KUKA KRL program: MyProgram_123().src

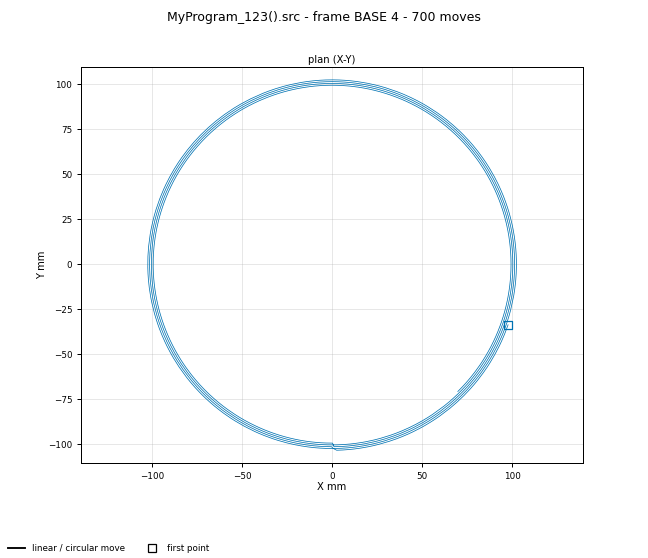
[picture p0: tool path of MyProgram_123().src in frame BASE 4, 700 of 700 moves have a stored position in this frame; points joined in program order, loops and branches not executed]
&ACCESS RVP
&REL 1
&PARAM TEMPLATE = C:\KRC\Roboter\Template\vorgabe
&PARAM EDITMASK = *
DEF MyProgram_123()
; ---- Setting reference (Base) ----
$BASE = BASE_DATA[4]

; --------------------------
; ---- Setting tool (TCP) ----
$TOOL = TOOL_DATA[3]
; --------------------------

$VEL.CP = VEL_APROX_PRINT
Startdeposition()
$VEL.CP = VEL_PRINT
LIN {X 97.6881,Y -33.6698,Z 103,A -23.787,B 24.9383,C -1.8145,E1 25.1507,E2 469.3571} C_DIS
LIN {X 95.781,Y -38.76,Z 103,A -26.6465,B 24.9385,C -1.8116,E1 25.1479,E2 472.2074} C_DIS
LIN {X 94.2157,Y -42.4228,Z 103,A -28.8922,B 24.939,C -1.8033,E1 25.1453,E2 474.4605} C_DIS
LIN {X 93.0003,Y -45.0257,Z 103,A -30.4605,B 24.9393,C -1.7995,E1 25.1435,E2 476.0292} C_DIS
LIN {X 90.4664,Y -49.9238,Z 103,A -33.4281,B 24.9397,C -1.7942,E1 25.1396,E2 478.9937} C_DIS
LIN {X 87.7675,Y -54.5272,Z 103,A -36.2353,B 24.9398,C -1.7919,E1 25.1357,E2 481.7919} C_DIS
LIN {X 86.0982,Y -57.1268,Z 103,A -37.9177,B 24.9401,C -1.7883,E1 25.1331,E2 483.4744} C_DIS
LIN {X 83.9825,Y -60.1936,Z 103,A -41.1362,B 24.9436,C -1.7353,E1 25.1277,E2 486.8023} C_DIS
LIN {X 80.9511,Y -64.2124,Z 103,A -42.7215,B 24.9408,C -1.7771,E1 25.1252,E2 488.2813} C_DIS
LIN {X 79.0718,Y -66.5134,Z 103,A -44.9977,B 24.9428,C -1.7469,E1 25.121,E2 490.6184} C_DIS
LIN {X 76.8006,Y -69.1233,Z 103,A -47.4937,B 24.9447,C -1.7186,E1 25.1163,E2 493.1703} C_DIS
LIN {X 73.2293,Y -72.8966,Z 103,A -49.516,B 24.9428,C -1.7463,E1 25.1125,E2 495.1185} C_DIS
LIN {X 69.1425,Y -76.7834,Z 103,A -52.3279,B 24.9425,C -1.7518,E1 25.1068,E2 497.9058} C_DIS
LIN {X 65.4366,Y -79.9649,Z 103,A -55.2445,B 24.9434,C -1.7371,E1 25.1005,E2 500.8457} C_DIS
LIN {X 59.791,Y -84.2698,Z 103,A -59.6873,B 24.9453,C -1.7083,E1 25.0905,E2 505.3406} C_DIS
LIN {X 56.834,Y -86.2913,Z 103,A -61.1986,B 24.9443,C -1.7235,E1 25.087,E2 506.811} C_DIS
LIN {X 54.8773,Y -87.5488,Z 103,A -63.0884,B 24.946,C -1.697,E1 25.0824,E2 508.7576} C_DIS
LIN {X 51.3153,Y -89.6831,Z 103,A -64.9043,B 24.9451,C -1.7122,E1 25.0781,E2 510.5318} C_DIS
LIN {X 48.7655,Y -91.0963,Z 103,A -67.0748,B 24.9466,C -1.6873,E1 25.0727,E2 512.7551} C_DIS
LIN {X 44.8398,Y -93.0897,Z 103,A -68.7427,B 24.9449,C -1.7142,E1 25.0687,E2 514.3551} C_DIS
LIN {X 42.065,Y -94.3769,Z 103,A -70.4455,B 24.9451,C -1.7113,E1 25.0643,E2 516.0605} C_DIS
LIN {X 38.6683,Y -95.8183,Z 103,A -72.4301,B 24.9451,C -1.7107,E1 25.0592,E2 518.0417} C_DIS
LIN {X 35.7045,Y -96.9617,Z 103,A -74.1219,B 24.9451,C -1.7111,E1 25.0548,E2 519.7289} C_DIS
LIN {X 31.6622,Y -98.3555,Z 103,A -76.9185,B 24.9464,C -1.6913,E1 25.0473,E2 522.567} C_DIS
LIN {X 25.8035,Y -100.0524,Z 103,A -79.9686,B 24.9458,C -1.7007,E1 25.0392,E2 525.5899} C_DIS
LIN {X 23.0245,Y -100.7284,Z 103,A -81.6681,B 24.9462,C -1.6947,E1 25.0345,E2 527.3012} C_DIS
LIN {X 20.0098,Y -101.3712,Z 103,A -83.5475,B 24.9467,C -1.6865,E1 25.0293,E2 529.1976} C_DIS
LIN {X 15.782,Y -102.1137,Z 103,A -85.6605,B 24.9461,C -1.6952,E1 25.0236,E2 531.288} C_DIS
LIN {X 12.1927,Y -102.6044,Z 103,A -87.6248,B 24.9461,C -1.6956,E1 25.0181,E2 533.2496} C_DIS
LIN {X 9.3968,Y -102.898,Z 103,A -89.2294,B 24.9463,C -1.693,E1 25.0136,E2 534.8595} C_DIS
LIN {X 5.8711,Y -103.1593,Z 103,A -91.1468,B 24.9463,C -1.6938,E1 25.0083,E2 536.7742} C_DIS
LIN {X 2.5701,Y -103.2946,Z 103,A -93.23,B 24.9469,C -1.6835,E1 25.0024,E2 538.8813} C_DIS
LIN {X 2.5701,Y -103.2946,Z 103,A -93.23,B 24.9469,C -1.6835,E1 25.0024,E2 538.8813} C_DIS
Enddeposition()
LIN {X 0.6764,Y -102.3239,Z 103,A -92.9796,B 24.9425,C -1.7511,E1 25.0036,E2 538.4707} C_DIS
Startdeposition()
$VEL.CP = VEL_PRINT
LIN {X 5.1299,Y -102.2014,Z 103,A -90.7138,B 24.9431,C -1.743,E1 25.0098,E2 536.2248} C_DIS
LIN {X 8.6252,Y -101.9657,Z 103,A -88.8428,B 24.9432,C -1.7404,E1 25.015,E2 534.3608} C_DIS
LIN {X 11.7328,Y -101.654,Z 103,A -87.1009,B 24.9432,C -1.7411,E1 25.0199,E2 532.6184} C_DIS
LIN {X 14.8311,Y -101.2492,Z 103,A -85.4205,B 24.9432,C -1.7396,E1 25.0245,E2 530.9431} C_DIS
LIN {X 18.0457,Y -100.725,Z 103,A -82.9702,B 24.9416,C -1.7658,E1 25.0314,E2 528.4332} C_DIS
LIN {X 21.7381,Y -99.9932,Z 103,A -81.7936,B 24.9439,C -1.7308,E1 25.0344,E2 527.341} C_DIS
LIN {X 25.3407,Y -99.1415,Z 103,A -78.7726,B 24.9412,C -1.7705,E1 25.0428,E2 524.2304} C_DIS
LIN {X 29.0621,Y -98.1151,Z 103,A -77.3225,B 24.943,C -1.7445,E1 25.0466,E2 522.8443} C_DIS
LIN {X 34.35,Y -96.3924,Z 103,A -74.2269,B 24.9428,C -1.7476,E1 25.0548,E2 519.7474} C_DIS
LIN {X 36.8204,Y -95.4766,Z 103,A -72.3941,B 24.9417,C -1.7639,E1 25.0596,E2 517.8799} C_DIS
LIN {X 40.9607,Y -93.7731,Z 103,A -70.1365,B 24.9421,C -1.7576,E1 25.0654,E2 515.6426} C_DIS
LIN {X 44.2148,Y -92.2835,Z 103,A -67.2701,B 24.9396,C -1.7958,E1 25.0728,E2 512.6934} C_DIS
LIN {X 48.6188,Y -90.0412,Z 103,A -65.4434,B 24.9418,C -1.7623,E1 25.0771,E2 510.9511} C_DIS
LIN {X 54.1864,Y -86.8044,Z 103,A -61.7565,B 24.9411,C -1.7721,E1 25.086,E2 507.2522} C_DIS
LIN {X 57.1319,Y -84.895,Z 103,A -59.6088,B 24.9404,C -1.7834,E1 25.091,E2 505.0849} C_DIS
LIN {X 62.2384,Y -81.2257,Z 103,A -56.2515,B 24.9404,C -1.7841,E1 25.0986,E2 501.738} C_DIS
LIN {X 64.8437,Y -79.1628,Z 103,A -53.7177,B 24.9382,C -1.8159,E1 25.1042,E2 499.1387} C_DIS
LIN {X 68.2158,Y -76.2743,Z 103,A -51.8271,B 24.9395,C -1.7971,E1 25.108,E2 497.3001} C_DIS
LIN {X 71.7921,Y -72.9185,Z 103,A -49.3095,B 24.9397,C -1.7943,E1 25.1131,E2 494.7995} C_DIS
LIN {X 74.8341,Y -69.7929,Z 103,A -46.659,B 24.9387,C -1.8089,E1 25.1182,E2 492.1259} C_DIS
LIN {X 79.0313,Y -65.0038,Z 103,A -43.5153,B 24.9392,C -1.8007,E1 25.1239,E2 489.0158} C_DIS
LIN {X 81.397,Y -62.0162,Z 103,A -40.7192,B 24.937,C -1.8339,E1 25.1288,E2 486.1545} C_DIS
LIN {X 83.3036,Y -59.4279,Z 103,A -39.15,B 24.9373,C -1.8293,E1 25.1313,E2 484.6039} C_DIS
LIN {X 86.6661,Y -54.4079,Z 103,A -36.2819,B 24.9381,C -1.8174,E1 25.1357,E2 481.7781} C_DIS
LIN {X 89.1842,Y -50.1743,Z 103,A -33.504,B 24.9375,C -1.8262,E1 25.1396,E2 478.9937} C_DIS
LIN {X 91.8425,Y -45.1248,Z 103,A -30.4364,B 24.9372,C -1.8303,E1 25.1436,E2 475.9326} C_DIS
LIN {X 93.9408,Y -40.5754,Z 103,A -27.3944,B 24.9359,C -1.8487,E1 25.1471,E2 472.8638} C_DIS
LIN {X 94.7427,Y -38.6652,Z 103,A -25.5293,B 24.9336,C -1.8818,E1 25.1492,E2 470.9309} C_DIS
LIN {X 96.193,Y -34.9014,Z 103,A -24.0542,B 24.9354,C -1.8559,E1 25.1505,E2 469.525} C_DIS
LIN {X 97.098,Y -32.3004,Z 103,A -22.1429,B 24.934,C -1.8762,E1 25.1523,E2 467.5768} C_DIS
LIN {X 98.3344,Y -28.3145,Z 103,A -20.2379,B 24.9348,C -1.8655,E1 25.1538,E2 465.7078} C_DIS
LIN {X 99.0904,Y -25.5398,Z 103,A -18.4059,B 24.9338,C -1.8799,E1 25.1551,E2 463.8524} C_DIS
LIN {X 100.8062,Y -17.5945,Z 103,A -13.9078,B 24.9329,C -1.8922,E1 25.1577,E2 459.3515} C_DIS
LIN {X 101.3003,Y -14.4716,Z 103,A -12.2038,B 24.9327,C -1.8951,E1 25.1584,E2 457.6507} C_DIS
LIN {X 101.6826,Y -11.4892,Z 103,A -10.5934,B 24.9325,C -1.8975,E1 25.1589,E2 456.0441} C_DIS
LIN {X 101.9596,Y -8.7015,Z 103,A -8.8579,B 24.9316,C -1.9095,E1 25.1593,E2 454.2906} C_DIS
LIN {X 102.2018,Y -5.1224,Z 103,A -6.8282,B 24.9311,C -1.9169,E1 25.1597,E2 452.2554} C_DIS
LIN {X 102.3205,Y -1.3896,Z 103,A -4.7846,B 24.9308,C -1.9217,E1 25.1597,E2 450.2128} C_DIS
LIN {X 102.3102,Y 1.9501,Z 103,A -3.0627,B 24.9308,C -1.9216,E1 25.1597,E2 448.5014} C_DIS
LIN {X 102.1959,Y 5.2298,Z 103,A -1.1425,B 24.9301,C -1.9309,E1 25.1595,E2 446.5705} C_DIS
LIN {X 101.9747,Y 8.5125,Z 103,A 0.6517,B 24.9298,C -1.9348,E1 25.1591,E2 444.7778} C_DIS
LIN {X 101.6184,Y 12.0368,Z 103,A 2.611,B 24.9294,C -1.9401,E1 25.1585,E2 442.8175} C_DIS
LIN {X 101.1396,Y 15.5552,Z 103,A 5.1372,B 24.9273,C -1.9689,E1 25.1575,E2 440.2382} C_DIS
LIN {X 100.4971,Y 19.2745,Z 103,A 6.4328,B 24.9293,C -1.9414,E1 25.1568,E2 439.0151} C_DIS
LIN {X 99.9925,Y 21.741,Z 103,A 8.6713,B 24.9265,C -1.9804,E1 25.1555,E2 436.6978} C_DIS
LIN {X 99.0888,Y 25.546,Z 103,A 10.6938,B 24.9265,C -1.9801,E1 25.1541,E2 434.6876} C_DIS
LIN {X 98.2038,Y 28.7626,Z 103,A 12.202,B 24.9272,C -1.9708,E1 25.1529,E2 433.21} C_DIS
LIN {X 97.3458,Y 31.543,Z 103,A 14.2272,B 24.9256,C -1.9922,E1 25.1512,E2 431.1459} C_DIS
LIN {X 96.1935,Y 34.9002,Z 103,A 16.1019,B 24.9255,C -1.9933,E1 25.1494,E2 429.2789} C_DIS
LIN {X 95.0448,Y 37.9205,Z 103,A 17.3004,B 24.927,C -1.9733,E1 25.1482,E2 428.1342} C_DIS
LIN {X 93.5446,Y 41.4843,Z 103,A 20.1796,B 24.9243,C -2.0091,E1 25.1449,E2 425.1863} C_DIS
LIN {X 92.0205,Y 44.7621,Z 103,A 21.5257,B 24.926,C -1.9868,E1 25.1434,E2 423.9001} C_DIS
LIN {X 90.0902,Y 48.5285,Z 103,A 24.9903,B 24.9221,C -2.0386,E1 25.1387,E2 420.3314} C_DIS
LIN {X 87.4182,Y 53.1905,Z 103,A 27.02,B 24.9245,C -2.0061,E1 25.1359,E2 418.3888} C_DIS
LIN {X 85.4679,Y 56.2709,Z 103,A 29.0531,B 24.9242,C -2.0111,E1 25.1328,E2 416.3542} C_DIS
LIN {X 83.4563,Y 59.2139,Z 103,A 31.0802,B 24.9237,C -2.0174,E1 25.1296,E2 414.3221} C_DIS
LIN {X 80.898,Y 62.6638,Z 103,A 33.6427,B 24.9227,C -2.0297,E1 25.1252,E2 411.7427} C_DIS
LIN {X 78.1456,Y 66.065,Z 103,A 35.6682,B 24.9236,C -2.0183,E1 25.1217,E2 409.7537} C_DIS
LIN {X 76.2538,Y 68.2388,Z 103,A 38.2863,B 24.9202,C -2.0629,E1 25.1167,E2 407.0418} C_DIS
LIN {X 72.9545,Y 71.7556,Z 103,A 40.1125,B 24.9225,C -2.0332,E1 25.1133,E2 405.2937} C_DIS
LIN {X 70.6983,Y 73.9805,Z 103,A 42.3393,B 24.9208,C -2.0552,E1 25.1087,E2 403.0241} C_DIS
LIN {X 67.1434,Y 77.2204,Z 103,A 44.6876,B 24.9215,C -2.0466,E1 25.1039,E2 400.7054} C_DIS
LIN {X 63.4119,Y 80.3126,Z 103,A 47.2997,B 24.9214,C -2.0476,E1 25.0982,E2 398.1007} C_DIS
LIN {X 60.5384,Y 82.5002,Z 103,A 49.2285,B 24.9214,C -2.0475,E1 25.0939,E2 396.1793} C_DIS
LIN {X 58.115,Y 84.2256,Z 103,A 51.0165,B 24.9208,C -2.0552,E1 25.0898,E2 394.3793} C_DIS
LIN {X 53.0343,Y 87.5131,Z 103,A 54.2793,B 24.9208,C -2.0554,E1 25.0822,E2 391.1263} C_DIS
LIN {X 50.3531,Y 89.0844,Z 103,A 56.6147,B 24.9187,C -2.0815,E1 25.0763,E2 388.7362} C_DIS
LIN {X 47.1208,Y 90.836,Z 103,A 58.0513,B 24.9205,C -2.0596,E1 25.0729,E2 387.3556} C_DIS
LIN {X 43.6056,Y 92.574,Z 103,A 61.0752,B 24.9177,C -2.095,E1 25.0651,E2 384.2557} C_DIS
LIN {X 39.5283,Y 94.3861,Z 103,A 62.7833,B 24.9199,C -2.0666,E1 25.0609,E2 382.6189} C_DIS
LIN {X 36.3047,Y 95.6721,Z 103,A 64.784,B 24.9196,C -2.0707,E1 25.0557,E2 380.6128} C_DIS
LIN {X 29.8111,Y 97.8914,Z 103,A 68.5164,B 24.9196,C -2.0696,E1 25.0458,E2 376.8903} C_DIS
LIN {X 26.1694,Y 98.9264,Z 103,A 70.7179,B 24.9193,C -2.0742,E1 25.0399,E2 374.6816} C_DIS
LIN {X 23.9575,Y 99.4852,Z 103,A 72.2118,B 24.9186,C -2.0833,E1 25.0358,E2 373.1682} C_DIS
LIN {X 19.7985,Y 100.3962,Z 103,A 74.4624,B 24.9189,C -2.0792,E1 25.0297,E2 370.9301} C_DIS
LIN {X 13.9711,Y 101.3714,Z 103,A 77.5904,B 24.9194,C -2.0733,E1 25.0211,E2 367.8192} C_DIS
LIN {X 10.1931,Y 101.8209,Z 103,A 79.8047,B 24.9191,C -2.0769,E1 25.0149,E2 365.598} C_DIS
LIN {X 7.1294,Y 102.0803,Z 103,A 81.5107,B 24.9191,C -2.0764,E1 25.0102,E2 363.894} C_DIS
LIN {X 3.8255,Y 102.2588,Z 103,A 83.4844,B 24.9188,C -2.0808,E1 25.0046,E2 361.9103} C_DIS
LIN {X 0.4603,Y 102.3279,Z 103,A 85.3216,B 24.919,C -2.0788,E1 24.9995,E2 360.0782} C_DIS
LIN {X -3.5745,Y 102.2672,Z 103,A 87.636,B 24.9188,C -2.0802,E1 24.9931,E2 357.7601} C_DIS
LIN {X -7.1158,Y 102.0813,Z 103,A 89.6197,B 24.9189,C -2.0794,E1 24.9875,E2 355.7778} C_DIS
LIN {X -10.6764,Y 101.7703,Z 103,A 91.525,B 24.9193,C -2.0748,E1 24.9823,E2 353.8824} C_DIS
LIN {X -14.2625,Y 101.33,Z 103,A 93.4881,B 24.9195,C -2.0713,E1 24.9768,E2 351.9261} C_DIS
LIN {X -16.901,Y 100.9234,Z 103,A 94.9678,B 24.9197,C -2.0697,E1 24.9728,E2 350.4489} C_DIS
LIN {X -22.928,Y 99.7271,Z 103,A 98.4341,B 24.9198,C -2.0677,E1 24.9633,E2 346.9833} C_DIS
LIN {X -27.1429,Y 98.6644,Z 103,A 100.741,B 24.9204,C -2.0606,E1 24.9571,E2 344.6899} C_DIS
LIN {X -31.3638,Y 97.4037,Z 103,A 104.032,B 24.9182,C -2.0882,E1 24.9481,E2 341.3275} C_DIS
LIN {X -35.1858,Y 96.0893,Z 103,A 105.5975,B 24.9205,C -2.0596,E1 24.9442,E2 339.8269} C_DIS
LIN {X -38.2688,Y 94.9041,Z 103,A 107.6339,B 24.9201,C -2.0639,E1 24.9389,E2 337.7758} C_DIS
LIN {X -45.384,Y 91.7141,Z 103,A 111.879,B 24.921,C -2.0528,E1 24.9281,E2 333.5467} C_DIS
LIN {X -50.8604,Y 88.7942,Z 103,A 115.7351,B 24.9204,C -2.0606,E1 24.9186,E2 329.6609} C_DIS
LIN {X -54.5538,Y 86.5749,Z 103,A 117.8765,B 24.9215,C -2.0463,E1 24.9136,E2 327.5469} C_DIS
LIN {X -59.8044,Y 83.0348,Z 103,A 121.2946,B 24.9224,C -2.0346,E1 24.9058,E2 324.1451} C_DIS
LIN {X -64.5863,Y 79.3715,Z 103,A 124.7343,B 24.9227,C -2.0298,E1 24.8982,E2 320.7043} C_DIS
LIN {X -68.7002,Y 75.8407,Z 103,A 127.839,B 24.9231,C -2.0253,E1 24.8916,E2 317.5981} C_DIS
LIN {X -73.1997,Y 71.5073,Z 103,A 131.2469,B 24.924,C -2.0137,E1 24.8849,E2 314.2035} C_DIS
LIN {X -76.7453,Y 67.6873,Z 103,A 134.119,B 24.9246,C -2.0047,E1 24.8795,E2 311.3401} C_DIS
LIN {X -80.3353,Y 63.3831,Z 103,A 137.4083,B 24.9249,C -2.0018,E1 24.8736,E2 308.0425} C_DIS
LIN {X -83.4011,Y 59.2913,Z 103,A 139.9123,B 24.9264,C -1.9815,E1 24.8695,E2 305.575} C_DIS
LIN {X -85.4174,Y 56.3476,Z 103,A 142.4607,B 24.9254,C -1.9952,E1 24.8654,E2 302.9812} C_DIS
LIN {X -87.5272,Y 53.0112,Z 103,A 144.4598,B 24.9264,C -1.9815,E1 24.8625,E2 301.0046} C_DIS
LIN {X -90.1139,Y 48.4849,Z 103,A 147.1082,B 24.9277,C -1.9635,E1 24.8589,E2 298.3852} C_DIS
LIN {X -92.3223,Y 44.134,Z 103,A 150.1271,B 24.9276,C -1.9653,E1 24.8551,E2 295.3457} C_DIS
LIN {X -93.56,Y 41.4495,Z 103,A 152.3955,B 24.9264,C -1.9818,E1 24.8525,E2 293.0257} C_DIS
LIN {X -94.8973,Y 38.2854,Z 103,A 153.677,B 24.9285,C -1.9535,E1 24.8512,E2 291.8046} C_DIS
LIN {X -95.6895,Y 36.2587,Z 103,A 155.0005,B 24.9285,C -1.9534,E1 24.8498,E2 290.4738} C_DIS
LIN {X -97.718,Y 30.3705,Z 103,A 158.5726,B 24.929,C -1.9454,E1 24.8467,E2 286.9004} C_DIS
LIN {X -98.7052,Y 26.9918,Z 103,A 160.5889,B 24.9294,C -1.9407,E1 24.8451,E2 284.8836} C_DIS
LIN {X -99.5938,Y 23.5051,Z 103,A 162.9118,B 24.9291,C -1.9451,E1 24.8436,E2 282.5367} C_DIS
LIN {X -100.4616,Y 19.4593,Z 103,A 164.887,B 24.9305,C -1.9258,E1 24.8425,E2 280.5958} C_DIS
LIN {X -100.9558,Y 16.7071,Z 103,A 166.5732,B 24.9305,C -1.9249,E1 24.8417,E2 278.9017} C_DIS
LIN {X -101.8577,Y 9.8159,Z 103,A 170.218,B 24.9321,C -1.9038,E1 24.8405,E2 275.2856} C_DIS
LIN {X -102.2389,Y 4.2897,Z 103,A 173.526,B 24.9323,C -1.9009,E1 24.8399,E2 271.9646} C_DIS
LIN {X -102.3141,Y -1.7362,Z 103,A 177.4161,B 24.9318,C -1.908,E1 24.8399,E2 268.0341} C_DIS
LIN {X -102.1965,Y -5.2188,Z 103,A 178.836,B 24.9335,C -1.8831,E1 24.8401,E2 266.6648} C_DIS
LIN {X -101.978,Y -8.4709,Z 103,A -178.4307,B 24.9317,C -1.9092,E1 24.8407,E2 263.853} C_DIS
LIN {X -101.4715,Y -13.2179,Z 103,A -176.6633,B 24.9345,C -1.8689,E1 24.8413,E2 262.1712} C_DIS
LIN {X -100.6597,Y -18.4088,Z 103,A -173.7406,B 24.9352,C -1.8589,E1 24.8426,E2 259.2549} C_DIS
LIN {X -100.1306,Y -21.1025,Z 103,A -170.8662,B 24.9322,C -1.9013,E1 24.8444,E2 256.2624} C_DIS
LIN {X -98.6728,Y -27.1118,Z 103,A -168.6846,B 24.9362,C -1.8454,E1 24.8458,E2 254.2016} C_DIS
LIN {X -98.0018,Y -29.4439,Z 103,A -167.0909,B 24.9359,C -1.8495,E1 24.8471,E2 252.5888} C_DIS
LIN {X -96.9171,Y -32.8369,Z 103,A -165.2409,B 24.9366,C -1.8385,E1 24.8487,E2 250.7546} C_DIS
LIN {X -95.9244,Y -35.6377,Z 103,A -163.5211,B 24.9369,C -1.8355,E1 24.8503,E2 249.0322} C_DIS
LIN {X -94.5224,Y -39.205,Z 103,A -160.7982,B 24.9359,C -1.8497,E1 24.8532,E2 246.2602} C_DIS
LIN {X -93.036,Y -42.6101,Z 103,A -159.2556,B 24.9376,C -1.8247,E1 24.855,E2 244.7688} C_DIS
LIN {X -91.6232,Y -45.5672,Z 103,A -156.9031,B 24.9367,C -1.8379,E1 24.8579,E2 242.3719} C_DIS
LIN {X -89.9679,Y -48.7539,Z 103,A -155.3643,B 24.9382,C -1.8156,E1 24.8599,E2 240.8782} C_DIS
LIN {X -88.1116,Y -52.0339,Z 103,A -153.2546,B 24.9386,C -1.81,E1 24.8628,E2 238.771} C_DIS
LIN {X -84.8933,Y -57.1348,Z 103,A -150.1412,B 24.9398,C -1.7918,E1 24.8675,E2 235.6853} C_DIS
LIN {X -80.6124,Y -63.0325,Z 103,A -145.9112,B 24.9402,C -1.7869,E1 24.8745,E2 231.4463} C_DIS
LIN {X -78.7267,Y -65.3704,Z 103,A -143.4235,B 24.9385,C -1.8121,E1 24.879,E2 228.8871} C_DIS
LIN {X -75.9857,Y -68.5383,Z 103,A -141.6205,B 24.9401,C -1.7871,E1 24.8823,E2 227.1357} C_DIS
LIN {X -73.5455,Y -71.1496,Z 103,A -139.6232,B 24.9404,C -1.7826,E1 24.8861,E2 225.1404} C_DIS
LIN {X -70.6353,Y -74.0412,Z 103,A -137.3889,B 24.9409,C -1.7755,E1 24.8906,E2 222.9137} C_DIS
LIN {X -68.025,Y -76.4452,Z 103,A -135.238,B 24.9408,C -1.7775,E1 24.8951,E2 220.7494} C_DIS
LIN {X -65.3778,Y -78.7205,Z 103,A -133.0319,B 24.9404,C -1.783,E1 24.8998,E2 218.5217} C_DIS
LIN {X -62.8231,Y -80.7753,Z 103,A -131.5254,B 24.9414,C -1.7676,E1 24.9031,E2 217.0463} C_DIS
LIN {X -60.0212,Y -82.8789,Z 103,A -128.8435,B 24.9399,C -1.7908,E1 24.9093,E2 214.2997} C_DIS
LIN {X -56.2195,Y -85.5018,Z 103,A -127.4971,B 24.9432,C -1.7409,E1 24.9122,E2 213.0676} C_DIS
LIN {X -54.054,Y -86.8872,Z 103,A -125.5812,B 24.9422,C -1.7562,E1 24.9168,E2 211.1093} C_DIS
LIN {X -48.7638,Y -89.9626,Z 103,A -122.1544,B 24.9425,C -1.7514,E1 24.9251,E2 207.6838} C_DIS
LIN {X -42.9756,Y -92.8672,Z 103,A -118.7297,B 24.9433,C -1.7394,E1 24.9336,E2 204.2786} C_DIS
LIN {X -40.7743,Y -93.8544,Z 103,A -117.1951,B 24.9429,C -1.7448,E1 24.9376,E2 202.7276} C_DIS
LIN {X -37.472,Y -95.2209,Z 103,A -114.2966,B 24.9408,C -1.7767,E1 24.9453,E2 199.7468} C_DIS
LIN {X -32.8026,Y -96.9287,Z 103,A -112.4237,B 24.9433,C -1.7398,E1 24.95,E2 197.958} C_DIS
LIN {X -29.8438,Y -97.8813,Z 103,A -110.4477,B 24.9428,C -1.7474,E1 24.9553,E2 195.9606} C_DIS
LIN {X -24.9006,Y -99.2546,Z 103,A -107.8718,B 24.9436,C -1.7344,E1 24.9622,E2 193.4117} C_DIS
LIN {X -20.7038,Y -100.2125,Z 103,A -104.7707,B 24.942,C -1.7597,E1 24.9709,E2 190.2466} C_DIS
LIN {X -16.9529,Y -100.9147,Z 103,A -103.2029,B 24.9434,C -1.7371,E1 24.975,E2 188.7309} C_DIS
LIN {X -13.4553,Y -101.4407,Z 103,A -101.1404,B 24.9433,C -1.7398,E1 24.9808,E2 186.6603} C_DIS
LIN {X -9.8351,Y -101.8559,Z 103,A -99.0775,B 24.9433,C -1.7405,E1 24.9865,E2 184.5946} C_DIS
LIN {X -6.3339,Y -102.1341,Z 103,A -97.1143,B 24.9433,C -1.7404,E1 24.992,E2 182.631} C_DIS
LIN {X -2.8924,Y -102.2882,Z 103,A -95.2071,B 24.9433,C -1.7398,E1 24.9973,E2 180.7249} C_DIS
LIN {X 0.6764,Y -102.3239,Z 103,A -92.9756,B 24.9426,C -1.7494,E1 25.0036,E2 178.4707} C_DIS
Enddeposition()
LIN {X 0.6764,Y -102.3239,Z 103,A -92.9756,B 24.9426,C -1.7494,E1 25.0036,E2 178.4707} C_DIS
Startdeposition()
$VEL.CP = VEL_PRINT
LIN {X -0.3386,Y -101.3312,Z 103,A -94.7636,B 24.9446,C -1.7199,E1 24.9984,E2 180.3285} C_DIS
LIN {X -3.8329,Y -101.2602,Z 103,A -96.7748,B 24.9446,C -1.7183,E1 24.9928,E2 182.3438} C_DIS
LIN {X -7.3254,Y -101.0675,Z 103,A -98.7847,B 24.9447,C -1.717,E1 24.9872,E2 184.3574} C_DIS
LIN {X -10.9296,Y -100.741,Z 103,A -100.8211,B 24.9447,C -1.7176,E1 24.9815,E2 186.3936} C_DIS
LIN {X -14.5352,Y -100.2839,Z 103,A -102.8494,B 24.9447,C -1.719,E1 24.9759,E2 188.42} C_DIS
LIN {X -20.0224,Y -99.3342,Z 103,A -105.8846,B 24.9443,C -1.7243,E1 24.9676,E2 191.4457} C_DIS
LIN {X -22.3901,Y -98.8277,Z 103,A -107.5854,B 24.945,C -1.7127,E1 24.9629,E2 193.1763} C_DIS
LIN {X -26.3791,Y -97.8376,Z 103,A -109.6967,B 24.9444,C -1.7219,E1 24.9572,E2 195.2688} C_DIS
LIN {X -29.6885,Y -96.8853,Z 103,A -111.6315,B 24.9444,C -1.7237,E1 24.952,E2 197.2026} C_DIS
LIN {X -33.0408,Y -95.7948,Z 103,A -114.1897,B 24.9455,C -1.7048,E1 24.9451,E2 199.8106} C_DIS
LIN {X -36.7283,Y -94.4415,Z 103,A -115.6228,B 24.9436,C -1.7355,E1 24.9416,E2 201.1737} C_DIS
LIN {X -39.2642,Y -93.4151,Z 103,A -117.3605,B 24.9439,C -1.7301,E1 24.937,E2 202.9281} C_DIS
LIN {X -42.5115,Y -91.9832,Z 103,A -120.1044,B 24.9455,C -1.7059,E1 24.9299,E2 205.7366} C_DIS
LIN {X -46.5487,Y -90.0084,Z 103,A -121.8135,B 24.9433,C -1.7389,E1 24.9259,E2 207.3717} C_DIS
LIN {X -51.2291,Y -87.4287,Z 103,A -124.7611,B 24.9429,C -1.7457,E1 24.9187,E2 210.3116} C_DIS
LIN {X -53.7614,Y -85.894,Z 103,A -126.6339,B 24.9432,C -1.7411,E1 24.9142,E2 212.2012} C_DIS
LIN {X -58.91,Y -82.4479,Z 103,A -130.1639,B 24.9429,C -1.7458,E1 24.906,E2 215.7318} C_DIS
LIN {X -61.326,Y -80.6691,Z 103,A -132.5258,B 24.9442,C -1.7253,E1 24.9007,E2 218.1511} C_DIS
LIN {X -64.5907,Y -78.0778,Z 103,A -134.1408,B 24.9422,C -1.7558,E1 24.8973,E2 219.6995} C_DIS
LIN {X -67.0495,Y -75.9782,Z 103,A -135.9027,B 24.9418,C -1.7617,E1 24.8936,E2 221.4544} C_DIS
LIN {X -70.2476,Y -73.0297,Z 103,A -138.4902,B 24.9418,C -1.7622,E1 24.8883,E2 224.0513} C_DIS
LIN {X -72.6365,Y -70.6555,Z 103,A -140.4872,B 24.9418,C -1.763,E1 24.8844,E2 226.0548} C_DIS
LIN {X -74.976,Y -68.168,Z 103,A -142.4724,B 24.9416,C -1.7654,E1 24.8806,E2 228.0431} C_DIS
LIN {X -78.1967,Y -64.4476,Z 103,A -145.275,B 24.9412,C -1.7711,E1 24.8755,E2 230.8448} C_DIS
LIN {X -82.8721,Y -58.3147,Z 103,A -149.4312,B 24.94,C -1.7888,E1 24.8686,E2 234.9787} C_DIS
LIN {X -86.0922,Y -53.4441,Z 103,A -152.9429,B 24.94,C -1.7901,E1 24.8632,E2 238.5052} C_DIS
LIN {X -87.8981,Y -50.418,Z 103,A -154.8899,B 24.9395,C -1.797,E1 24.8605,E2 240.4459} C_DIS
LIN {X -90.0561,Y -46.4554,Z 103,A -157.4723,B 24.9391,C -1.8029,E1 24.8571,E2 243.0278} C_DIS
LIN {X -91.608,Y -43.3175,Z 103,A -159.8265,B 24.9396,C -1.7956,E1 24.8542,E2 245.4121} C_DIS
LIN {X -93.5259,Y -39.0013,Z 103,A -162.2542,B 24.9385,C -1.8116,E1 24.8516,E2 247.8152} C_DIS
LIN {X -94.7887,Y -35.8211,Z 103,A -164.1136,B 24.9379,C -1.8198,E1 24.8497,E2 249.6654} C_DIS
LIN {X -96.0821,Y -32.1918,Z 103,A -166.3532,B 24.9376,C -1.8242,E1 24.8476,E2 251.9073} C_DIS
LIN {X -97.2137,Y -28.5939,Z 103,A -168.4919,B 24.9372,C -1.8304,E1 24.8459,E2 254.0434} C_DIS
LIN {X -98.8398,Y -22.338,Z 103,A -171.9745,B 24.936,C -1.8475,E1 24.8436,E2 257.5056} C_DIS
LIN {X -99.4475,Y -19.4508,Z 103,A -173.8041,B 24.936,C -1.8472,E1 24.8425,E2 259.3467} C_DIS
LIN {X -100.3589,Y -14.0073,Z 103,A -176.6942,B 24.9348,C -1.8649,E1 24.8413,E2 262.2119} C_DIS
LIN {X -100.8742,Y -9.6203,Z 103,A -179.5164,B 24.935,C -1.8618,E1 24.8404,E2 265.0583} C_DIS
LIN {X -101.1089,Y -6.7124,Z 103,A 178.0701,B 24.9364,C -1.8415,E1 24.84,E2 267.5347} C_DIS
LIN {X -101.3139,Y -1.8842,Z 103,A 175.6823,B 24.935,C -1.8618,E1 24.8398,E2 269.8886} C_DIS
LIN {X -101.3194,Y 1.5802,Z 103,A 174.1684,B 24.9335,C -1.883,E1 24.8398,E2 271.361} C_DIS
LIN {X -101.1243,Y 6.4851,Z 103,A 171.0038,B 24.9338,C -1.8789,E1 24.8403,E2 274.5544} C_DIS
LIN {X -100.3123,Y 14.3355,Z 103,A 166.9532,B 24.9318,C -1.9071,E1 24.8416,E2 278.5619} C_DIS
LIN {X -99.3008,Y 20.185,Z 103,A 163.4507,B 24.9314,C -1.913,E1 24.8433,E2 282.0713} C_DIS
LIN {X -98.4442,Y 24.0165,Z 103,A 161.3289,B 24.9306,C -1.9233,E1 24.8446,E2 284.1807} C_DIS
LIN {X -97.6401,Y 27.1064,Z 103,A 159.4015,B 24.9306,C -1.9249,E1 24.846,E2 286.1155} C_DIS
LIN {X -96.601,Y 30.6051,Z 103,A 156.6601,B 24.9317,C -1.9087,E1 24.8484,E2 288.9115} C_DIS
LIN {X -95.2138,Y 34.6755,Z 103,A 154.9014,B 24.9295,C -1.9388,E1 24.85,E2 290.6083} C_DIS
LIN {X -93.5038,Y 39.0537,Z 103,A 152.2304,B 24.929,C -1.9465,E1 24.8527,E2 293.2759} C_DIS
LIN {X -92.0934,Y 42.2746,Z 103,A 150.1852,B 24.9287,C -1.9505,E1 24.8551,E2 295.3226} C_DIS
LIN {X -89.7998,Y 46.9484,Z 103,A 147.3265,B 24.9278,C -1.9622,E1 24.8586,E2 298.169} C_DIS
LIN {X -87.7943,Y 50.5987,Z 103,A 144.9371,B 24.9274,C -1.9679,E1 24.8619,E2 300.5574} C_DIS
LIN {X -85.7868,Y 53.9329,Z 103,A 141.8396,B 24.9292,C -1.9439,E1 24.8666,E2 303.7279} C_DIS
LIN {X -83.0518,Y 58.0561,Z 103,A 139.9676,B 24.9263,C -1.9829,E1 24.8694,E2 305.5161} C_DIS
LIN {X -80.6207,Y 61.3896,Z 103,A 137.6284,B 24.9258,C -1.9889,E1 24.8733,E2 307.8521} C_DIS
LIN {X -77.1377,Y 65.7101,Z 103,A 134.3977,B 24.9254,C -1.994,E1 24.879,E2 311.0858} C_DIS
LIN {X -73.5211,Y 69.7344,Z 103,A 131.4118,B 24.9247,C -2.0042,E1 24.8846,E2 314.0606} C_DIS
LIN {X -69.2582,Y 73.9689,Z 103,A 127.9781,B 24.9242,C -2.0111,E1 24.8914,E2 317.4923} C_DIS
LIN {X -65.4143,Y 77.3898,Z 103,A 125.0271,B 24.9238,C -2.0162,E1 24.8976,E2 320.4427} C_DIS
LIN {X -61.5007,Y 80.5352,Z 103,A 121.895,B 24.9241,C -2.0122,E1 24.9045,E2 323.5961} C_DIS
LIN {X -57.6106,Y 83.3615,Z 103,A 119.1064,B 24.9238,C -2.0153,E1 24.9109,E2 326.3868} C_DIS
LIN {X -53.6314,Y 85.9751,Z 103,A 116.0773,B 24.9243,C -2.0087,E1 24.9181,E2 329.4412} C_DIS
LIN {X -50.2044,Y 88.0209,Z 103,A 114.5771,B 24.922,C -2.0391,E1 24.9216,E2 330.8736} C_DIS
LIN {X -48.2093,Y 89.1287,Z 103,A 113.0732,B 24.9224,C -2.0338,E1 24.9253,E2 332.3943} C_DIS
LIN {X -45.0496,Y 90.7667,Z 103,A 111.1152,B 24.922,C -2.039,E1 24.9301,E2 334.3452} C_DIS
LIN {X -38.936,Y 93.5534,Z 103,A 107.5769,B 24.9209,C -2.0539,E1 24.9391,E2 337.8567} C_DIS
LIN {X -35.3504,Y 94.967,Z 103,A 104.7731,B 24.9224,C -2.0346,E1 24.9465,E2 340.7123} C_DIS
LIN {X -30.1192,Y 96.7517,Z 103,A 102.3399,B 24.9202,C -2.0631,E1 24.9528,E2 343.0823} C_DIS
LIN {X -27.777,Y 97.4501,Z 103,A 100.6241,B 24.921,C -2.0526,E1 24.9575,E2 344.8259} C_DIS
LIN {X -24.7648,Y 98.2598,Z 103,A 98.6419,B 24.9215,C -2.0465,E1 24.9629,E2 346.8254} C_DIS
LIN {X -20.8453,Y 99.1646,Z 103,A 96.1713,B 24.9218,C -2.0415,E1 24.9696,E2 349.3111} C_DIS
LIN {X -16.5708,Y 99.9674,Z 103,A 94.1541,B 24.9205,C -2.0593,E1 24.9751,E2 351.288} C_DIS
LIN {X -13.7239,Y 100.3992,Z 103,A 92.352,B 24.9209,C -2.054,E1 24.9801,E2 353.1041} C_DIS
LIN {X -10.3269,Y 100.8041,Z 103,A 90.5443,B 24.9204,C -2.0597,E1 24.9851,E2 354.8994} C_DIS
LIN {X -6.7781,Y 101.1045,Z 103,A 88.5271,B 24.9204,C -2.0605,E1 24.9907,E2 356.9157} C_DIS
LIN {X -3.2856,Y 101.2783,Z 103,A 86.4841,B 24.9205,C -2.0587,E1 24.9964,E2 358.9633} C_DIS
LIN {X 0.0115,Y 101.3332,Z 103,A 84.542,B 24.9207,C -2.0562,E1 25.0018,E2 360.9113} C_DIS
LIN {X 3.4907,Y 101.272,Z 103,A 82.6206,B 24.9206,C -2.0582,E1 25.0072,E2 362.8277} C_DIS
LIN {X 6.9232,Y 101.0947,Z 103,A 80.6928,B 24.9206,C -2.0588,E1 25.0126,E2 364.7533} C_DIS
LIN {X 11.0188,Y 100.7316,Z 103,A 78.3906,B 24.9205,C -2.0593,E1 25.019,E2 367.0527} C_DIS
LIN {X 13.3667,Y 100.4465,Z 103,A 76.1079,B 24.9232,C -2.0241,E1 25.0255,E2 369.4169} C_DIS
LIN {X 18.6879,Y 99.5944,Z 103,A 74.0962,B 24.9203,C -2.0613,E1 25.0308,E2 371.3384} C_DIS
LIN {X 23.2163,Y 98.6369,Z 103,A 71.4973,B 24.9203,C -2.0607,E1 25.0379,E2 373.9353} C_DIS
LIN {X 26.581,Y 97.7831,Z 103,A 69.4517,B 24.9207,C -2.0563,E1 25.0434,E2 375.988} C_DIS
LIN {X 30.0466,Y 96.7742,Z 103,A 66.8065,B 24.9226,C -2.0321,E1 25.0506,E2 378.6859} C_DIS
LIN {X 33.8728,Y 95.5029,Z 103,A 65.0869,B 24.9211,C -2.0512,E1 25.055,E2 380.3569} C_DIS
LIN {X 37.2515,Y 94.236,Z 103,A 63.0178,B 24.9213,C -2.0481,E1 25.0604,E2 382.4287} C_DIS
LIN {X 44.5408,Y 91.0189,Z 103,A 57.7879,B 24.9238,C -2.0154,E1 25.0738,E2 387.7229} C_DIS
LIN {X 48.8347,Y 88.7894,Z 103,A 55.7801,B 24.922,C -2.0394,E1 25.0786,E2 389.6681} C_DIS
LIN {X 52.0269,Y 86.9571,Z 103,A 53.3826,B 24.9232,C -2.0242,E1 25.0845,E2 392.0942} C_DIS
LIN {X 54.7466,Y 85.2693,Z 103,A 51.7306,B 24.9229,C -2.0274,E1 25.0883,E2 393.7332} C_DIS
LIN {X 57.8942,Y 83.1644,Z 103,A 49.8837,B 24.9223,C -2.0353,E1 25.0925,E2 395.5553} C_DIS
LIN {X 60.871,Y 81.0109,Z 103,A 47.9319,B 24.9223,C -2.0365,E1 25.0969,E2 397.4971} C_DIS
LIN {X 63.0688,Y 79.3125,Z 103,A 46.1625,B 24.923,C -2.0259,E1 25.1008,E2 399.2852} C_DIS
LIN {X 65.8855,Y 76.9883,Z 103,A 44.2582,B 24.9229,C -2.0282,E1 25.1049,E2 401.1767} C_DIS
LIN {X 68.6799,Y 74.5062,Z 103,A 42.3324,B 24.9226,C -2.0313,E1 25.1088,E2 403.0873} C_DIS
LIN {X 70.4953,Y 72.7909,Z 103,A 40.642,B 24.9237,C -2.0174,E1 25.1123,E2 404.8036} C_DIS
LIN {X 72.9785,Y 70.3007,Z 103,A 38.2536,B 24.9252,C -1.9974,E1 25.117,E2 407.2289} C_DIS
LIN {X 75.2786,Y 67.8328,Z 103,A 37.0497,B 24.9234,C -2.0209,E1 25.1192,E2 408.3722} C_DIS
LIN {X 78.2259,Y 64.4125,Z 103,A 33.6216,B 24.9265,C -1.9804,E1 25.1255,E2 411.8803} C_DIS
LIN {X 80.759,Y 61.2064,Z 103,A 31.8778,B 24.9252,C -1.9971,E1 25.1284,E2 413.5764} C_DIS
LIN {X 82.7569,Y 58.477,Z 103,A 30.0448,B 24.9253,C -1.9955,E1 25.1313,E2 415.4044} C_DIS
LIN {X 84.5804,Y 55.8051,Z 103,A 28.222,B 24.9257,C -1.991,E1 25.1342,E2 417.2286} C_DIS
LIN {X 86.5926,Y 52.6287,Z 103,A 25.6013,B 24.9275,C -1.9658,E1 25.1381,E2 419.8956} C_DIS
LIN {X 88.4349,Y 49.4705,Z 103,A 23.6319,B 24.9277,C -1.964,E1 25.1408,E2 421.8588} C_DIS
LIN {X 90.0343,Y 46.498,Z 103,A 22.3699,B 24.9262,C -1.9846,E1 25.1423,E2 423.0656} C_DIS
LIN {X 92.2517,Y 41.9259,Z 103,A 19.5002,B 24.9267,C -1.9766,E1 25.1458,E2 425.9386} C_DIS
LIN {X 93.3633,Y 39.3872,Z 103,A 17.7424,B 24.9276,C -1.9644,E1 25.1478,E2 427.7157} C_DIS
LIN {X 95.7416,Y 33.1925,Z 103,A 13.9641,B 24.9285,C -1.9523,E1 25.1515,E2 431.5015} C_DIS
LIN {X 96.8244,Y 29.8848,Z 103,A 11.5044,B 24.9304,C -1.9266,E1 25.1536,E2 434.0079} C_DIS
LIN {X 97.8905,Y 26.1832,Z 103,A 9.6233,B 24.93,C -1.9318,E1 25.1549,E2 435.8657} C_DIS
LIN {X 99.1516,Y 20.9121,Z 103,A 6.731,B 24.9302,C -1.9293,E1 25.1567,E2 438.7474} C_DIS
LIN {X 100.1705,Y 15.2959,Z 103,A 4.1747,B 24.929,C -1.9465,E1 25.1579,E2 441.2481} C_DIS
LIN {X 100.4954,Y 12.9895,Z 103,A 2.3678,B 24.9307,C -1.9223,E1 25.1586,E2 443.1014} C_DIS
LIN {X 100.8996,Y 9.3442,Z 103,A 0.2929,B 24.9312,C -1.9156,E1 25.1592,E2 445.1797} C_DIS
LIN {X 101.1665,Y 5.7822,Z 103,A -1.7103,B 24.9316,C -1.9098,E1 25.1596,E2 447.1847} C_DIS
LIN {X 101.3082,Y 2.1938,Z 103,A -3.7362,B 24.9321,C -1.9035,E1 25.1598,E2 449.2136} C_DIS
LIN {X 101.3259,Y -1.2141,Z 103,A -5.7157,B 24.9327,C -1.8951,E1 25.1598,E2 451.201} C_DIS
LIN {X 101.2317,Y -4.496,Z 103,A -7.5313,B 24.933,C -1.8908,E1 25.1596,E2 453.016} C_DIS
LIN {X 100.9978,Y -8.2172,Z 103,A -9.5404,B 24.9332,C -1.888,E1 25.1592,E2 455.0198} C_DIS
LIN {X 100.6617,Y -11.6319,Z 103,A -11.5157,B 24.9337,C -1.8803,E1 25.1586,E2 457.0016} C_DIS
LIN {X 100.211,Y -15.0339,Z 103,A -13.4743,B 24.9342,C -1.8733,E1 25.1578,E2 458.9652} C_DIS
LIN {X 99.5499,Y -18.9187,Z 103,A -16.6707,B 24.9374,C -1.827,E1 25.1561,E2 462.2519} C_DIS
LIN {X 98.3485,Y -24.4088,Z 103,A -18.6393,B 24.9347,C -1.8657,E1 25.1549,E2 464.1179} C_DIS
LIN {X 97.3662,Y -28.073,Z 103,A -20.7768,B 24.9352,C -1.8592,E1 25.1534,E2 466.2584} C_DIS
LIN {X 96.5798,Y -30.6704,Z 103,A -22.316,B 24.9356,C -1.8542,E1 25.1521,E2 467.8008} C_DIS
LIN {X 95.7531,Y -33.1597,Z 103,A -23.9372,B 24.9363,C -1.8439,E1 25.1506,E2 469.437} C_DIS
LIN {X 94.2532,Y -37.2077,Z 103,A -26.4696,B 24.937,C -1.8326,E1 25.1481,E2 471.9818} C_DIS
LIN {X 91.9873,Y -42.5025,Z 103,A -29.3166,B 24.9366,C -1.8394,E1 25.145,E2 474.7975} C_DIS
LIN {X 90.8246,Y -44.9327,Z 103,A -31.7625,B 24.9394,C -1.7975,E1 25.1418,E2 477.3292} C_DIS
LIN {X 88.8729,Y -48.6809,Z 103,A -33.554,B 24.9383,C -1.8145,E1 25.1395,E2 479.0711} C_DIS
LIN {X 86.4869,Y -52.8025,Z 103,A -35.9382,B 24.938,C -1.8192,E1 25.1362,E2 481.4318} C_DIS
LIN {X 84.3138,Y -56.2089,Z 103,A -38.4839,B 24.9391,C -1.8021,E1 25.1323,E2 484.0051} C_DIS
LIN {X 82.6248,Y -58.6622,Z 103,A -40.0857,B 24.9392,C -1.8008,E1 25.1297,E2 485.6023} C_DIS
LIN {X 80.6073,Y -61.4066,Z 103,A -41.8691,B 24.9392,C -1.8013,E1 25.1268,E2 487.3759} C_DIS
LIN {X 78.7563,Y -63.7612,Z 103,A -43.7044,B 24.9399,C -1.7911,E1 25.1235,E2 489.2268} C_DIS
LIN {X 75.6595,Y -67.4073,Z 103,A -46.8052,B 24.9414,C -1.7682,E1 25.1178,E2 492.3675} C_DIS
LIN {X 73.3951,Y -69.8683,Z 103,A -48.1645,B 24.9403,C -1.7847,E1 25.1153,E2 493.6819} C_DIS
LIN {X 71.3401,Y -71.963,Z 103,A -49.902,B 24.9408,C -1.7775,E1 25.1118,E2 495.4289} C_DIS
LIN {X 67.6149,Y -75.4737,Z 103,A -53.1042,B 24.942,C -1.7584,E1 25.1052,E2 498.6632} C_DIS
LIN {X 64.6932,Y -77.9926,Z 103,A -54.9907,B 24.9416,C -1.7652,E1 25.1012,E2 500.5264} C_DIS
LIN {X 60.17,Y -81.5337,Z 103,A -58.3038,B 24.9422,C -1.7557,E1 25.0939,E2 503.8501} C_DIS
LIN {X 57.433,Y -83.484,Z 103,A -60.1997,B 24.9425,C -1.752,E1 25.0895,E2 505.7482} C_DIS
LIN {X 55.0983,Y -85.0436,Z 103,A -61.7004,B 24.9425,C -1.7523,E1 25.086,E2 507.2431} C_DIS
LIN {X 50.6285,Y -87.7772,Z 103,A -64.2885,B 24.9418,C -1.7616,E1 25.0799,E2 509.8012} C_DIS
LIN {X 45.7351,Y -90.4242,Z 103,A -67.9636,B 24.9436,C -1.7353,E1 25.0707,E2 513.5281} C_DIS
LIN {X 42.8245,Y -91.8375,Z 103,A -69.5829,B 24.9432,C -1.7406,E1 25.0667,E2 515.1307} C_DIS
LIN {X 39.6159,Y -93.2669,Z 103,A -71.4594,B 24.9432,C -1.7419,E1 25.0619,E2 516.9996} C_DIS
LIN {X 37.5778,Y -94.1078,Z 103,A -72.934,B 24.9438,C -1.7312,E1 25.058,E2 518.4961} C_DIS
LIN {X 34.2203,Y -95.3798,Z 103,A -75.2508,B 24.9447,C -1.7174,E1 25.0519,E2 520.8407} C_DIS
LIN {X 29.4523,Y -96.9585,Z 103,A -78.1147,B 24.945,C -1.7131,E1 25.0442,E2 523.7095} C_DIS
LIN {X 26.2982,Y -97.8594,Z 103,A -79.4509,B 24.9438,C -1.7311,E1 25.0408,E2 525.001} C_DIS
LIN {X 23.9258,Y -98.4663,Z 103,A -80.9902,B 24.9443,C -1.7237,E1 25.0365,E2 526.5554} C_DIS
LIN {X 18.4861,Y -99.6325,Z 103,A -84.0738,B 24.9443,C -1.7234,E1 25.0281,E2 529.6361} C_DIS
LIN {X 15.316,Y -100.1674,Z 103,A -85.8009,B 24.9443,C -1.7255,E1 25.0234,E2 531.3564} C_DIS
LIN {X 11.8551,Y -100.6355,Z 103,A -87.7933,B 24.9443,C -1.7236,E1 25.0178,E2 533.3518} C_DIS
LIN {X 8.3629,Y -100.9861,Z 103,A -89.8053,B 24.9445,C -1.7215,E1 25.0122,E2 535.3677} C_DIS
LIN {X 5.4554,Y -101.1845,Z 103,A -91.4835,B 24.9445,C -1.7196,E1 25.0075,E2 537.0495} C_DIS
LIN {X 1.0493,Y -101.3269,Z 103,A -93.8969,B 24.9445,C -1.7218,E1 25.0008,E2 539.4573} C_DIS
LIN {X 1.0493,Y -101.3269,Z 103,A -93.8969,B 24.9445,C -1.7218,E1 25.0008,E2 539.4573} C_DIS
Enddeposition()
LIN {X 0.6699,Y -100.3286,Z 103,A -93.9374,B 24.9429,C -1.7459,E1 25.0008,E2 539.4406} C_DIS
Startdeposition()
$VEL.CP = VEL_PRINT
LIN {X 3.0141,Y -100.2888,Z 103,A -92.0127,B 24.9414,C -1.7684,E1 25.0064,E2 537.4629} C_DIS
LIN {X 6.3812,Y -100.1317,Z 103,A -90.045,B 24.9412,C -1.7708,E1 25.0119,E2 535.4903} C_DIS
LIN {X 9.9135,Y -99.8445,Z 103,A -88.0153,B 24.9412,C -1.7721,E1 25.0175,E2 533.4588} C_DIS
LIN {X 13.1077,Y -99.4744,Z 103,A -86.1721,B 24.941,C -1.7735,E1 25.0227,E2 531.6135} C_DIS
LIN {X 16.4154,Y -98.9822,Z 103,A -84.3162,B 24.941,C -1.7729,E1 25.0278,E2 529.761} C_DIS
LIN {X 18.9297,Y -98.5322,Z 103,A -82.1336,B 24.9391,C -1.8022,E1 25.0339,E2 527.5115} C_DIS
LIN {X 23.2948,Y -97.5937,Z 103,A -80.2351,B 24.9407,C -1.7792,E1 25.0389,E2 525.6701} C_DIS
LIN {X 26.6919,Y -96.72,Z 103,A -78.0762,B 24.9401,C -1.7874,E1 25.0448,E2 523.4953} C_DIS
LIN {X 32.324,Y -94.985,Z 103,A -74.9452,B 24.9405,C -1.7823,E1 25.0531,E2 520.3822} C_DIS
LIN {X 35.6175,Y -93.7994,Z 103,A -72.9007,B 24.9402,C -1.7868,E1 25.0584,E2 518.3314} C_DIS
LIN {X 38.6519,Y -92.5908,Z 103,A -71.0974,B 24.9402,C -1.787,E1 25.0631,E2 516.5316} C_DIS
LIN {X 43.0257,Y -90.6418,Z 103,A -68.5591,B 24.9404,C -1.7835,E1 25.0695,E2 514.008} C_DIS
LIN {X 46.7943,Y -88.7537,Z 103,A -65.4823,B 24.9383,C -1.8141,E1 25.0773,E2 510.8674} C_DIS
LIN {X 49.9061,Y -87.042,Z 103,A -63.9677,B 24.9395,C -1.7973,E1 25.0809,E2 509.397} C_DIS
LIN {X 53.0999,Y -85.1312,Z 103,A -61.855,B 24.9392,C -1.8008,E1 25.0859,E2 507.2827} C_DIS
LIN {X 55.6527,Y -83.4862,Z 103,A -59.8514,B 24.9383,C -1.8149,E1 25.0907,E2 505.2523} C_DIS
LIN {X 62.2985,Y -78.65,Z 103,A -55.4261,B 24.9383,C -1.814,E1 25.1005,E2 500.8449} C_DIS
LIN {X 64.9039,Y -76.5143,Z 103,A -53.597,B 24.9383,C -1.8145,E1 25.1044,E2 499.0217} C_DIS
LIN {X 67.0139,Y -74.6731,Z 103,A -51.8217,B 24.9375,C -1.8253,E1 25.1082,E2 497.2279} C_DIS
LIN {X 69.9087,Y -71.9711,Z 103,A -49.6046,B 24.9373,C -1.8289,E1 25.1127,E2 495.0115} C_DIS
LIN {X 72.4695,Y -69.3916,Z 103,A -47.6172,B 24.9372,C -1.8305,E1 25.1165,E2 493.0289} C_DIS
LIN {X 74.9687,Y -66.6836,Z 103,A -45.5225,B 24.9369,C -1.8355,E1 25.1205,E2 490.9318} C_DIS
LIN {X 77.1831,Y -64.1068,Z 103,A -43.5893,B 24.9365,C -1.8403,E1 25.1239,E2 488.9961} C_DIS
LIN {X 79.5094,Y -61.1979,Z 103,A -41.536,B 24.9363,C -1.843,E1 25.1275,E2 486.9461} C_DIS
LIN {X 82.1041,Y -57.6722,Z 103,A -37.9801,B 24.9328,C -1.893,E1 25.1334,E2 483.2893} C_DIS
LIN {X 85.1506,Y -53.0688,Z 103,A -35.9546,B 24.9354,C -1.8558,E1 25.1363,E2 481.3618} C_DIS
LIN {X 86.6997,Y -50.5018,Z 103,A -34.0808,B 24.9346,C -1.8673,E1 25.139,E2 479.4704} C_DIS
LIN {X 88.1403,Y -47.9398,Z 103,A -31.9019,B 24.9328,C -1.8928,E1 25.1419,E2 477.2429} C_DIS
LIN {X 89.9508,Y -44.4498,Z 103,A -30.2218,B 24.934,C -1.8763,E1 25.144,E2 475.6106} C_DIS
LIN {X 91.5284,Y -41.1034,Z 103,A -27.9719,B 24.9332,C -1.8883,E1 25.1466,E2 473.3446} C_DIS
LIN {X 93.7569,Y -35.7297,Z 103,A -24.805,B 24.9329,C -1.8922,E1 25.1499,E2 470.1861} C_DIS
LIN {X 94.9116,Y -32.5417,Z 103,A -22.8234,B 24.9323,C -1.9001,E1 25.1517,E2 468.197} C_DIS
LIN {X 95.9362,Y -29.3818,Z 103,A -21.101,B 24.9324,C -1.8989,E1 25.1532,E2 466.4871} C_DIS
LIN {X 96.8021,Y -26.3879,Z 103,A -19.2743,B 24.9319,C -1.9065,E1 25.1545,E2 464.6531} C_DIS
LIN {X 97.683,Y -22.9144,Z 103,A -17.2329,B 24.9314,C -1.9128,E1 25.1559,E2 462.6086} C_DIS
LIN {X 98.2588,Y -20.3011,Z 103,A -15.0824,B 24.9292,C -1.9433,E1 25.1572,E2 460.3986} C_DIS
LIN {X 99.0251,Y -16.1589,Z 103,A -13.2617,B 24.9304,C -1.9269,E1 25.158,E2 458.6272} C_DIS
LIN {X 99.5362,Y -12.6309,Z 103,A -11.3343,B 24.9302,C -1.9291,E1 25.1587,E2 456.7062} C_DIS
LIN {X 99.9071,Y -9.246,Z 103,A -9.4412,B 24.9299,C -1.9332,E1 25.1592,E2 454.8144} C_DIS
LIN {X 100.1534,Y -6.0381,Z 103,A -7.4804,B 24.9291,C -1.9442,E1 25.1596,E2 452.8394} C_DIS
LIN {X 100.3101,Y -2.2259,Z 103,A -5.3801,B 24.9289,C -1.9481,E1 25.1598,E2 450.7426} C_DIS
LIN {X 100.3288,Y 1.1636,Z 103,A -3.3897,B 24.9282,C -1.9565,E1 25.1598,E2 448.744} C_DIS
LIN {X 100.2151,Y 4.9232,Z 103,A -1.3508,B 24.928,C -1.959,E1 25.1595,E2 446.7114} C_DIS
LIN {X 100.011,Y 8.0448,Z 103,A 0.4184,B 24.9277,C -1.964,E1 25.1592,E2 444.9408} C_DIS
LIN {X 99.6324,Y 11.8461,Z 103,A 2.6551,B 24.927,C -1.9732,E1 25.1585,E2 442.6956} C_DIS
LIN {X 99.2167,Y 14.937,Z 103,A 4.9548,B 24.925,C -2.0001,E1 25.1575,E2 440.3461} C_DIS
LIN {X 98.5559,Y 18.8062,Z 103,A 6.5707,B 24.9264,C -1.9815,E1 25.1567,E2 438.7834} C_DIS
LIN {X 97.8149,Y 22.3434,Z 103,A 8.329,B 24.9268,C -1.9755,E1 25.1557,E2 437.0496} C_DIS
LIN {X 96.6017,Y 27.1126,Z 103,A 11.4952,B 24.9251,C -1.9986,E1 25.1534,E2 433.8472} C_DIS
LIN {X 95.5564,Y 30.5938,Z 103,A 13.5152,B 24.9248,C -2.0026,E1 25.1518,E2 431.8293} C_DIS
LIN {X 94.454,Y 33.848,Z 103,A 15.2995,B 24.9249,C -2.0012,E1 25.1501,E2 430.0583} C_DIS
LIN {X 93.1445,Y 37.3008,Z 103,A 17.5359,B 24.9241,C -2.0125,E1 25.1479,E2 427.8075} C_DIS
LIN {X 92.0521,Y 39.9169,Z 103,A 19.1563,B 24.9237,C -2.0173,E1 25.1461,E2 426.1848} C_DIS
LIN {X 90.0331,Y 44.2838,Z 103,A 21.8063,B 24.9234,C -2.0211,E1 25.1429,E2 423.54} C_DIS
LIN {X 88.7134,Y 46.8707,Z 103,A 23.4628,B 24.9231,C -2.0256,E1 25.1408,E2 421.8816} C_DIS
LIN {X 85.8982,Y 51.8508,Z 103,A 26.7709,B 24.9223,C -2.036,E1 25.1362,E2 418.5661} C_DIS
LIN {X 84.1834,Y 54.592,Z 103,A 28.5234,B 24.9222,C -2.0371,E1 25.1336,E2 416.8199} C_DIS
LIN {X 82.341,Y 57.3314,Z 103,A 30.5553,B 24.9214,C -2.0478,E1 25.1303,E2 414.7728} C_DIS
LIN {X 80.6183,Y 59.7321,Z 103,A 33.1385,B 24.9182,C -2.0879,E1 25.1259,E2 412.107} C_DIS
LIN {X 77.3054,Y 63.9597,Z 103,A 35.219,B 24.9208,C -2.0556,E1 25.1224,E2 410.1126} C_DIS
LIN {X 75.0043,Y 66.644,Z 103,A 36.9805,B 24.9212,C -2.05,E1 25.1192,E2 408.3722} C_DIS
LIN {X 72.8757,Y 68.9648,Z 103,A 39.0016,B 24.9202,C -2.0628,E1 25.1153,E2 406.3297} C_DIS
LIN {X 70.4982,Y 71.3927,Z 103,A 40.9438,B 24.9199,C -2.0671,E1 25.1115,E2 404.3857} C_DIS
LIN {X 67.8175,Y 73.944,Z 103,A 42.9597,B 24.9199,C -2.0676,E1 25.1074,E2 402.3769} C_DIS
LIN {X 65.3071,Y 76.1708,Z 103,A 44.9539,B 24.9193,C -2.0744,E1 25.1031,E2 400.3744} C_DIS
LIN {X 62.7256,Y 78.3119,Z 103,A 46.93,B 24.9188,C -2.0804,E1 25.0989,E2 398.3918} C_DIS
LIN {X 59.7081,Y 80.6359,Z 103,A 49.1885,B 24.9183,C -2.0875,E1 25.0938,E2 396.1244} C_DIS
LIN {X 56.6156,Y 82.8356,Z 103,A 51.5564,B 24.9174,C -2.099,E1 25.0883,E2 393.7375} C_DIS
LIN {X 51.2649,Y 86.249,Z 103,A 54.8153,B 24.9181,C -2.0903,E1 25.0807,E2 390.5095} C_DIS
LIN {X 48.0116,Y 88.1013,Z 103,A 56.6784,B 24.9187,C -2.0827,E1 25.0762,E2 388.6699} C_DIS
LIN {X 44.9287,Y 89.7134,Z 103,A 58.915,B 24.9177,C -2.0949,E1 25.0706,E2 386.4107} C_DIS
LIN {X 41.7688,Y 91.2285,Z 103,A 61.365,B 24.9161,C -2.1145,E1 25.0643,E2 383.9204} C_DIS
LIN {X 38.7217,Y 92.5614,Z 103,A 62.8838,B 24.9171,C -2.1019,E1 25.0604,E2 382.435} C_DIS
LIN {X 35.3005,Y 93.9194,Z 103,A 64.9954,B 24.917,C -2.1044,E1 25.0549,E2 380.3223} C_DIS
LIN {X 32.53,Y 94.9156,Z 103,A 66.802,B 24.9165,C -2.1106,E1 25.0501,E2 378.5045} C_DIS
LIN {X 28.459,Y 96.2133,Z 103,A 68.9497,B 24.9172,C -2.1013,E1 25.0445,E2 376.3826} C_DIS
LIN {X 25.083,Y 97.1482,Z 103,A 71.0425,B 24.9168,C -2.1061,E1 25.0388,E2 374.2817} C_DIS
LIN {X 21.7104,Y 97.9576,Z 103,A 73.1554,B 24.9163,C -2.1121,E1 25.033,E2 372.1574} C_DIS
LIN {X 17.9751,Y 98.711,Z 103,A 75.18,B 24.9167,C -2.1073,E1 25.0275,E2 370.1466} C_DIS
LIN {X 15.5064,Y 99.1287,Z 103,A 76.923,B 24.9157,C -2.1196,E1 25.0226,E2 368.3763} C_DIS
LIN {X 11.9218,Y 99.6236,Z 103,A 79.2501,B 24.9149,C -2.1297,E1 25.0161,E2 366.0268} C_DIS
LIN {X 8.0386,Y 100.0115,Z 103,A 80.8725,B 24.9167,C -2.1072,E1 25.0118,E2 364.4587} C_DIS
LIN {X 4.6557,Y 100.2266,Z 103,A 82.7787,B 24.9168,C -2.1061,E1 25.0064,E2 362.556} C_DIS
LIN {X 1.341,Y 100.3263,Z 103,A 84.7687,B 24.9166,C -2.1094,E1 25.0009,E2 360.5584} C_DIS
LIN {X -2.0494,Y 100.3133,Z 103,A 86.7523,B 24.9164,C -2.1107,E1 24.9953,E2 358.5717} C_DIS
LIN {X -5.6295,Y 100.176,Z 103,A 88.7554,B 24.9166,C -2.1084,E1 24.9897,E2 356.5734} C_DIS
LIN {X -9.2517,Y 99.9066,Z 103,A 90.8091,B 24.9168,C -2.1067,E1 24.984,E2 354.5229} C_DIS
LIN {X -12.9711,Y 99.4921,Z 103,A 92.8982,B 24.917,C -2.1037,E1 24.9783,E2 352.4395} C_DIS
LIN {X -16.5753,Y 98.9554,Z 103,A 94.8019,B 24.9176,C -2.0958,E1 24.9731,E2 350.5527} C_DIS
LIN {X -21.0235,Y 98.1074,Z 103,A 97.6159,B 24.9171,C -2.102,E1 24.9653,E2 347.7211} C_DIS
LIN {X -24.4592,Y 97.3085,Z 103,A 99.6485,B 24.9172,C -2.1007,E1 24.9598,E2 345.6887} C_DIS
LIN {X -27.6474,Y 96.4502,Z 103,A 101.5768,B 24.9172,C -2.1003,E1 24.9546,E2 343.7584} C_DIS
LIN {X -31.014,Y 95.4205,Z 103,A 103.4497,B 24.9178,C -2.093,E1 24.9496,E2 341.8995} C_DIS
LIN {X -35.1758,Y 93.9666,Z 103,A 106.001,B 24.918,C -2.091,E1 24.9429,E2 339.3478} C_DIS
LIN {X -38.0994,Y 92.8194,Z 103,A 107.7252,B 24.9184,C -2.0861,E1 24.9385,E2 337.6315} C_DIS
LIN {X -41.6207,Y 91.2953,Z 103,A 110.1077,B 24.9181,C -2.0896,E1 24.9324,E2 335.2349} C_DIS
LIN {X -45.0765,Y 89.6402,Z 103,A 112.3635,B 24.9182,C -2.0885,E1 24.9267,E2 332.9758} C_DIS
LIN {X -48.5314,Y 87.817,Z 103,A 114.5161,B 24.9187,C -2.0819,E1 24.9214,E2 330.8327} C_DIS
LIN {X -51.3325,Y 86.209,Z 103,A 116.1933,B 24.9194,C -2.0728,E1 24.9174,E2 329.1724} C_DIS
LIN {X -54.2709,Y 84.3895,Z 103,A 118.1998,B 24.9196,C -2.0702,E1 24.9127,E2 327.1656} C_DIS
LIN {X -58.6067,Y 81.4392,Z 103,A 121.8238,B 24.9184,C -2.0863,E1 24.9043,E2 323.4909} C_DIS
LIN {X -61.4633,Y 79.3048,Z 103,A 123.1119,B 24.9207,C -2.0558,E1 24.9016,E2 322.2708} C_DIS
LIN {X -63.7946,Y 77.4425,Z 103,A 125.0115,B 24.9205,C -2.0589,E1 24.8974,E2 320.3568} C_DIS
LIN {X -66.5691,Y 75.0713,Z 103,A 127.2283,B 24.9205,C -2.0588,E1 24.8927,E2 318.1315} C_DIS
LIN {X -69.1702,Y 72.6826,Z 103,A 129.133,B 24.9212,C -2.0501,E1 24.8889,E2 316.2395} C_DIS
LIN {X -71.9441,Y 69.9368,Z 103,A 131.4347,B 24.9214,C -2.0473,E1 24.8843,E2 313.9349} C_DIS
LIN {X -74.4416,Y 67.2724,Z 103,A 133.5886,B 24.9216,C -2.0444,E1 24.8803,E2 311.7784} C_DIS
LIN {X -76.8243,Y 64.5386,Z 103,A 135.6346,B 24.9221,C -2.0382,E1 24.8766,E2 309.7378} C_DIS
LIN {X -79.2177,Y 61.5765,Z 103,A 137.5873,B 24.9231,C -2.0249,E1 24.8732,E2 307.8078} C_DIS
LIN {X -80.8803,Y 59.3743,Z 103,A 139.403,B 24.9228,C -2.0288,E1 24.8701,E2 305.9739} C_DIS
LIN {X -84.9685,Y 53.3604,Z 103,A 143.58,B 24.9236,C -2.018,E1 24.8637,E2 301.8018} C_DIS
LIN {X -86.7223,Y 50.4625,Z 103,A 145.8342,B 24.9232,C -2.0234,E1 24.8604,E2 299.5231} C_DIS
LIN {X -89.5357,Y 45.2819,Z 103,A 148.9725,B 24.9246,C -2.0057,E1 24.8564,E2 296.4104} C_DIS
LIN {X -90.843,Y 42.5975,Z 103,A 150.6102,B 24.9251,C -1.9983,E1 24.8544,E2 294.7815} C_DIS
LIN {X -92.2643,Y 39.4268,Z 103,A 152.702,B 24.9253,C -1.9959,E1 24.8521,E2 292.6838} C_DIS
LIN {X -93.2965,Y 36.9153,Z 103,A 154.244,B 24.9257,C -1.9909,E1 24.8505,E2 291.1452} C_DIS
LIN {X -94.9245,Y 32.5036,Z 103,A 156.8795,B 24.9264,C -1.9808,E1 24.848,E2 288.5187} C_DIS
LIN {X -95.9806,Y 29.2385,Z 103,A 158.9596,B 24.9266,C -1.9788,E1 24.8463,E2 286.4315} C_DIS
LIN {X -96.874,Y 26.1218,Z 103,A 160.6768,B 24.9274,C -1.9684,E1 24.845,E2 284.7292} C_DIS
LIN {X -97.596,Y 23.2851,Z 103,A 162.4106,B 24.9276,C -1.9652,E1 24.8439,E2 282.9929} C_DIS
LIN {X -98.4068,Y 19.5805,Z 103,A 164.8359,B 24.9275,C -1.9671,E1 24.8425,E2 280.5487} C_DIS
LIN {X -99.1129,Y 15.6089,Z 103,A 166.9078,B 24.9286,C -1.9518,E1 24.8415,E2 278.5009} C_DIS
LIN {X -99.4618,Y 13.2049,Z 103,A 168.7443,B 24.9278,C -1.9626,E1 24.8409,E2 276.6276} C_DIS
LIN {X -99.8551,Y 9.8097,Z 103,A 170.3708,B 24.9291,C -1.9452,E1 24.8404,E2 275.0329} C_DIS
LIN {X -100.2205,Y 4.7956,Z 103,A 173.2586,B 24.9297,C -1.9365,E1 24.8399,E2 272.1485} C_DIS
LIN {X -100.3349,Y -0.1393,Z 103,A 176.1147,B 24.9303,C -1.9287,E1 24.8398,E2 269.2938} C_DIS
LIN {X -100.2183,Y -4.8481,Z 103,A 178.7787,B 24.9309,C -1.9192,E1 24.8401,E2 266.6365} C_DIS
LIN {X -99.941,Y -8.8792,Z 103,A -178.4219,B 24.9303,C -1.9287,E1 24.8407,E2 263.7977} C_DIS
LIN {X -99.5411,Y -12.5931,Z 103,A -176.8381,B 24.9321,C -1.9031,E1 24.8412,E2 262.2654} C_DIS
LIN {X -99.2249,Y -14.884,Z 103,A -175.3702,B 24.9321,C -1.9039,E1 24.8418,E2 260.7868} C_DIS
LIN {X -98.6153,Y -18.498,Z 103,A -173.3029,B 24.9326,C -1.8965,E1 24.8429,E2 258.7249} C_DIS
LIN {X -97.8626,Y -22.1367,Z 103,A -171.2601,B 24.9332,C -1.8872,E1 24.8441,E2 256.6922} C_DIS
LIN {X -96.8999,Y -26.026,Z 103,A -168.9995,B 24.9338,C -1.8793,E1 24.8456,E2 254.4374} C_DIS
LIN {X -96.0408,Y -29.0406,Z 103,A -167.2318,B 24.9342,C -1.8731,E1 24.847,E2 252.6743} C_DIS
LIN {X -95.0882,Y -32.018,Z 103,A -165.3462,B 24.9344,C -1.8712,E1 24.8486,E2 250.7824} C_DIS
LIN {X -93.8766,Y -35.4135,Z 103,A -163.3706,B 24.935,C -1.8623,E1 24.8505,E2 248.8169} C_DIS
LIN {X -92.5233,Y -38.8122,Z 103,A -160.6259,B 24.9338,C -1.8789,E1 24.8535,E2 246.0174} C_DIS
LIN {X -91.0163,Y -42.2252,Z 103,A -159.011,B 24.9355,C -1.8549,E1 24.8553,E2 244.4507} C_DIS
LIN {X -89.3987,Y -45.55,Z 103,A -156.8892,B 24.9359,C -1.8494,E1 24.858,E2 242.3307} C_DIS
LIN {X -87.6569,Y -48.8181,Z 103,A -154.8051,B 24.9364,C -1.8426,E1 24.8608,E2 240.2518} C_DIS
LIN {X -86.0014,Y -51.681,Z 103,A -152.7851,B 24.9364,C -1.8421,E1 24.8636,E2 238.2225} C_DIS
LIN {X -83.5091,Y -55.618,Z 103,A -150.1304,B 24.9369,C -1.835,E1 24.8677,E2 235.5713} C_DIS
LIN {X -81.4385,Y -58.6077,Z 103,A -148.2136,B 24.9376,C -1.8242,E1 24.8707,E2 233.6708} C_DIS
LIN {X -80.1942,Y -60.2977,Z 103,A -146.5422,B 24.9367,C -1.8379,E1 24.8736,E2 231.9588} C_DIS
LIN {X -77.2219,Y -64.0602,Z 103,A -144.122,B 24.9379,C -1.8202,E1 24.8778,E2 229.5695} C_DIS
LIN {X -74.7639,Y -66.9125,Z 103,A -142.0208,B 24.9383,C -1.8136,E1 24.8816,E2 227.4746} C_DIS
LIN {X -72.3835,Y -69.4809,Z 103,A -139.9833,B 24.9386,C -1.8105,E1 24.8856,E2 225.4354} C_DIS
LIN {X -69.7918,Y -72.0838,Z 103,A -137.8503,B 24.9388,C -1.8074,E1 24.8898,E2 223.301} C_DIS
LIN {X -67.0728,Y -74.6203,Z 103,A -135.7596,B 24.9391,C -1.802,E1 24.8941,E2 221.2148} C_DIS
LIN {X -64.4795,Y -76.8734,Z 103,A -133.9702,B 24.9398,C -1.792,E1 24.8979,E2 219.442} C_DIS
LIN {X -61.2289,Y -79.4854,Z 103,A -131.3918,B 24.9396,C -1.7947,E1 24.9035,E2 216.8478} C_DIS
LIN {X -58.8955,Y -81.2309,Z 103,A -128.7671,B 24.9375,C -1.8265,E1 24.9097,E2 214.1381} C_DIS
LIN {X -54.563,Y -84.202,Z 103,A -126.6597,B 24.94,C -1.7894,E1 24.9144,E2 212.1122} C_DIS
LIN {X -51.5438,Y -86.0841,Z 103,A -124.5626,B 24.94,C -1.7887,E1 24.9194,E2 210.0102} C_DIS
LIN {X -48.1176,Y -88.0438,Z 103,A -122.4638,B 24.9406,C -1.78,E1 24.9245,E2 207.926} C_DIS
LIN {X -45.2079,Y -89.5735,Z 103,A -120.6519,B 24.9409,C -1.7752,E1 24.929,E2 206.1206} C_DIS
LIN {X -41.8978,Y -91.1687,Z 103,A -118.4688,B 24.9409,C -1.7759,E1 24.9345,E2 203.9304} C_DIS
LIN {X -38.7831,Y -92.5355,Z 103,A -116.4105,B 24.9407,C -1.778,E1 24.9398,E2 201.8621} C_DIS
LIN {X -35.4831,Y -93.8503,Z 103,A -114.2852,B 24.9407,C -1.7797,E1 24.9454,E2 199.7284} C_DIS
LIN {X -32.079,Y -95.0677,Z 103,A -112.3793,B 24.9411,C -1.7721,E1 24.9503,E2 197.8368} C_DIS
LIN {X -29.0245,Y -96.0456,Z 103,A -110.4823,B 24.9411,C -1.7732,E1 24.9554,E2 195.9341} C_DIS
LIN {X -25.5526,Y -97.0275,Z 103,A -108.5945,B 24.9416,C -1.7655,E1 24.9605,E2 194.0616} C_DIS
LIN {X -21.7934,Y -97.9395,Z 103,A -106.1996,B 24.9412,C -1.7712,E1 24.967,E2 191.6497} C_DIS
LIN {X -16.0022,Y -99.0513,Z 103,A -102.812,B 24.9412,C -1.7708,E1 24.9763,E2 188.2597} C_DIS
LIN {X -12.612,Y -99.5386,Z 103,A -100.8769,B 24.9413,C -1.7696,E1 24.9817,E2 186.3259} C_DIS
LIN {X -9.1488,Y -99.9161,Z 103,A -99.0137,B 24.9416,C -1.7647,E1 24.9868,E2 184.4733} C_DIS
LIN {X -6.0381,Y -100.1534,Z 103,A -97.0692,B 24.9412,C -1.7709,E1 24.9923,E2 182.5135} C_DIS
LIN {X -2.4102,Y -100.3067,Z 103,A -94.9851,B 24.9412,C -1.7715,E1 24.9981,E2 180.4276} C_DIS
LIN {X 0.6699,Y -100.3286,Z 103,A -93.9357,B 24.9429,C -1.7452,E1 25.0009,E2 179.4406} C_DIS
Enddeposition()
LIN {X 0.6699,Y -100.3286,Z 103,A -93.9357,B 24.9429,C -1.7452,E1 25.0009,E2 179.4406} C_DIS
Startdeposition()
$VEL.CP = VEL_PRINT
LIN {X 0.2227,Y -99.3372,Z 103,A -94.5688,B 24.9427,C -1.7486,E1 24.9991,E2 180.0655} C_DIS
LIN {X -3.2417,Y -99.284,Z 103,A -96.3777,B 24.9423,C -1.7553,E1 24.9941,E2 181.8588} C_DIS
LIN {X -6.0904,Y -99.1517,Z 103,A -98.0227,B 24.9423,C -1.7552,E1 24.9895,E2 183.5046} C_DIS
LIN {X -8.5182,Y -98.9726,Z 103,A -99.6325,B 24.9428,C -1.7477,E1 24.985,E2 185.1328} C_DIS
LIN {X -11.7503,Y -98.6395,Z 103,A -101.3012,B 24.9422,C -1.7555,E1 24.9804,E2 186.7842} C_DIS
LIN {X -14.577,Y -98.2632,Z 103,A -103.1239,B 24.9426,C -1.7493,E1 24.9753,E2 188.623} C_DIS
LIN {X -17.7978,Y -97.7295,Z 103,A -104.8299,B 24.9422,C -1.7564,E1 24.9707,E2 190.3138} C_DIS
LIN {X -20.1731,Y -97.267,Z 103,A -106.2831,B 24.9422,C -1.7549,E1 24.9667,E2 191.7723} C_DIS
LIN {X -23.384,Y -96.5453,Z 103,A -108.2263,B 24.9423,C -1.7542,E1 24.9614,E2 193.7196} C_DIS
LIN {X -26.1064,Y -95.845,Z 103,A -109.8109,B 24.9422,C -1.7565,E1 24.9571,E2 195.3011} C_DIS
LIN {X -28.8437,Y -95.0588,Z 103,A -111.5608,B 24.9424,C -1.7538,E1 24.9524,E2 197.0604} C_DIS
LIN {X -31.9174,Y -94.0696,Z 103,A -113.3199,B 24.942,C -1.759,E1 24.9478,E2 198.8104} C_DIS
LIN {X -34.6191,Y -93.111,Z 103,A -115.0837,B 24.9422,C -1.7565,E1 24.9431,E2 200.5837} C_DIS
LIN {X -37.571,Y -91.9577,Z 103,A -116.7643,B 24.9417,C -1.7635,E1 24.9388,E2 202.2512} C_DIS
LIN {X -40.255,Y -90.8167,Z 103,A -118.4381,B 24.9416,C -1.7656,E1 24.9345,E2 203.924} C_DIS
LIN {X -42.8654,Y -89.6123,Z 103,A -120.1985,B 24.9416,C -1.7639,E1 24.93,E2 205.6928} C_DIS
LIN {X -45.7136,Y -88.195,Z 103,A -122.1071,B 24.9417,C -1.7636,E1 24.9253,E2 207.6073} C_DIS
LIN {X -48.4988,Y -86.6928,Z 103,A -123.7964,B 24.9412,C -1.7709,E1 24.9212,E2 209.2841} C_DIS
LIN {X -51.0733,Y -85.2036,Z 103,A -125.6564,B 24.9414,C -1.7683,E1 24.9167,E2 211.1561} C_DIS
LIN {X -53.8214,Y -83.4929,Z 103,A -127.4433,B 24.941,C -1.774,E1 24.9125,E2 212.935} C_DIS
LIN {X -56.2264,Y -81.8944,Z 103,A -129.0318,B 24.9407,C -1.7793,E1 24.9088,E2 214.5161} C_DIS
LIN {X -58.0295,Y -80.6258,Z 103,A -130.3311,B 24.9406,C -1.7805,E1 24.9058,E2 215.8171} C_DIS
LIN {X -60.6288,Y -78.6888,Z 103,A -132.2364,B 24.9404,C -1.7826,E1 24.9016,E2 217.7243} C_DIS
LIN {X -63.085,Y -76.7354,Z 103,A -134.1891,B 24.9406,C -1.781,E1 24.8973,E2 219.6881} C_DIS
LIN {X -65.8033,Y -74.4182,Z 103,A -136.2956,B 24.9404,C -1.7834,E1 24.8929,E2 221.7973} C_DIS
LIN {X -68.5039,Y -71.9399,Z 103,A -138.4141,B 24.9401,C -1.7875,E1 24.8886,E2 223.9145} C_DIS
LIN {X -71.1007,Y -69.3746,Z 103,A -140.5313,B 24.9398,C -1.7916,E1 24.8844,E2 226.031} C_DIS
LIN {X -73.6014,Y -66.7156,Z 103,A -142.6466,B 24.9395,C -1.7959,E1 24.8804,E2 228.1453} C_DIS
LIN {X -76.0025,Y -63.9668,Z 103,A -144.7422,B 24.9392,C -1.8011,E1 24.8766,E2 230.238} C_DIS
LIN {X -78.2042,Y -61.2541,Z 103,A -146.5244,B 24.9383,C -1.8138,E1 24.8735,E2 231.9983} C_DIS
LIN {X -79.5478,Y -59.4975,Z 103,A -147.8542,B 24.9383,C -1.8151,E1 24.8713,E2 233.3314} C_DIS
LIN {X -80.9775,Y -57.5366,Z 103,A -149.2615,B 24.938,C -1.8183,E1 24.869,E2 234.7379} C_DIS
LIN {X -82.359,Y -55.541,Z 103,A -150.6693,B 24.9378,C -1.8216,E1 24.8668,E2 236.1449} C_DIS
LIN {X -83.886,Y -53.209,Z 103,A -152.2905,B 24.9376,C -1.8253,E1 24.8643,E2 237.7655} C_DIS
LIN {X -85.418,Y -50.7108,Z 103,A -154.0658,B 24.9374,C -1.8269,E1 24.8617,E2 239.5461} C_DIS
LIN {X -86.9263,Y -48.0807,Z 103,A -155.9347,B 24.9374,C -1.8276,E1 24.8592,E2 241.4232} C_DIS
LIN {X -88.5435,Y -45.0319,Z 103,A -157.8058,B 24.9367,C -1.8371,E1 24.8568,E2 243.2815} C_DIS
LIN {X -89.9765,Y -42.0956,Z 103,A -159.753,B 24.9365,C -1.8403,E1 24.8544,E2 245.2317} C_DIS
LIN {X -91.1409,Y -39.5114,Z 103,A -161.2727,B 24.9359,C -1.8488,E1 24.8527,E2 246.7395} C_DIS
LIN {X -92.2312,Y -36.899,Z 103,A -162.9337,B 24.9357,C -1.8526,E1 24.851,E2 248.4007} C_DIS
LIN {X -93.2555,Y -34.2232,Z 103,A -164.7009,B 24.9356,C -1.8536,E1 24.8492,E2 250.1754} C_DIS
LIN {X -94.3263,Y -31.1558,Z 103,A -166.6484,B 24.9354,C -1.8567,E1 24.8475,E2 252.1265} C_DIS
LIN {X -95.2885,Y -28.0697,Z 103,A -168.3599,B 24.9346,C -1.8675,E1 24.8461,E2 253.8223} C_DIS
LIN {X -96.0566,Y -25.3233,Z 103,A -170.0235,B 24.9343,C -1.8718,E1 24.8449,E2 255.4851} C_DIS
LIN {X -96.7469,Y -22.5356,Z 103,A -171.7839,B 24.9343,C -1.8735,E1 24.8437,E2 257.2518} C_DIS
LIN {X -97.4301,Y -19.3784,Z 103,A -173.5591,B 24.9336,C -1.8822,E1 24.8427,E2 259.0168} C_DIS
LIN {X -97.8753,Y -16.9873,Z 103,A -175.1417,B 24.9336,C -1.8806,E1 24.8419,E2 260.6126} C_DIS
LIN {X -98.3763,Y -13.7807,Z 103,A -176.8262,B 24.9328,C -1.8928,E1 24.8412,E2 262.2781} C_DIS
LIN {X -98.736,Y -10.9234,Z 103,A -178.5253,B 24.9326,C -1.8967,E1 24.8407,E2 263.9779} C_DIS
LIN {X -99.0062,Y -8.0988,Z 103,A 179.7228,B 24.9325,C -1.8982,E1 24.8402,E2 265.7368} C_DIS
LIN {X -99.2181,Y -4.8884,Z 103,A 177.7936,B 24.9322,C -1.9017,E1 24.8399,E2 267.6693} C_DIS
LIN {X -99.3226,Y -1.6759,Z 103,A 176.0416,B 24.9315,C -1.911,E1 24.8398,E2 269.4096} C_DIS
LIN {X -99.3315,Y 1.1534,Z 103,A 174.4427,B 24.9311,C -1.9173,E1 24.8398,E2 271.0031} C_DIS
LIN {X -99.2841,Y 3.2378,Z 103,A 173.1748,B 24.931,C -1.9191,E1 24.8399,E2 272.2744} C_DIS
LIN {X -99.1223,Y 6.5249,Z 103,A 171.2213,B 24.9306,C -1.9234,E1 24.8402,E2 274.2294} C_DIS
LIN {X -98.8986,Y 9.3204,Z 103,A 169.6916,B 24.9301,C -1.9315,E1 24.8406,E2 275.749} C_DIS
LIN {X -98.6379,Y 11.7637,Z 103,A 168.2643,B 24.9298,C -1.9357,E1 24.841,E2 277.1747} C_DIS
LIN {X -98.2626,Y 14.5807,Z 103,A 166.4486,B 24.9298,C -1.9352,E1 24.8417,E2 279.0026} C_DIS
LIN {X -97.7364,Y 17.7597,Z 103,A 164.7419,B 24.929,C -1.9461,E1 24.8425,E2 280.6932} C_DIS
LIN {X -97.2667,Y 20.1743,Z 103,A 163.2535,B 24.9288,C -1.9484,E1 24.8434,E2 282.185} C_DIS
LIN {X -96.5504,Y 23.3632,Z 103,A 161.3124,B 24.9285,C -1.9525,E1 24.8446,E2 284.1276} C_DIS
LIN {X -95.8499,Y 26.0883,Z 103,A 159.7221,B 24.9281,C -1.9587,E1 24.8457,E2 285.7124} C_DIS
LIN {X -95.0634,Y 28.8284,Z 103,A 157.9599,B 24.928,C -1.96,E1 24.8471,E2 287.4817} C_DIS
LIN {X -94.0741,Y 31.9041,Z 103,A 156.1882,B 24.9273,C -1.9689,E1 24.8487,E2 289.2424} C_DIS
LIN {X -93.2009,Y 34.3728,Z 103,A 154.5287,B 24.9273,C -1.9686,E1 24.8503,E2 290.9119} C_DIS
LIN {X -91.9301,Y 37.6387,Z 103,A 152.633,B 24.9266,C -1.979,E1 24.8522,E2 292.7935} C_DIS
LIN {X -90.6424,Y 40.642,Z 103,A 150.6932,B 24.9263,C -1.9829,E1 24.8544,E2 294.7347} C_DIS
LIN {X -89.3559,Y 43.399,Z 103,A 149.0419,B 24.9256,C -1.9915,E1 24.8563,E2 296.3743} C_DIS
LIN {X -88.1499,Y 45.8004,Z 103,A 147.3133,B 24.9257,C -1.9902,E1 24.8586,E2 298.1153} C_DIS
LIN {X -86.6241,Y 48.622,Z 103,A 145.6072,B 24.925,C -2.0004,E1 24.8608,E2 299.8062} C_DIS
LIN {X -85.4145,Y 50.7166,Z 103,A 144.2031,B 24.9247,C -2.0041,E1 24.8628,E2 301.2087} C_DIS
LIN {X -83.9335,Y 53.1347,Z 103,A 142.5556,B 24.9244,C -2.0083,E1 24.8652,E2 302.8545} C_DIS
LIN {X -82.3832,Y 55.5053,Z 103,A 140.8014,B 24.9244,C -2.0089,E1 24.868,E2 304.6161} C_DIS
LIN {X -80.5125,Y 58.1884,Z 103,A 139.0139,B 24.9237,C -2.0174,E1 24.8708,E2 306.3922} C_DIS
LIN {X -79.1503,Y 60.0268,Z 103,A 137.6659,B 24.9235,C -2.02,E1 24.8731,E2 307.7404} C_DIS
LIN {X -77.1663,Y 62.555,Z 103,A 135.7134,B 24.9234,C -2.0216,E1 24.8765,E2 309.6983} C_DIS
LIN {X -74.8193,Y 65.344,Z 103,A 133.5995,B 24.923,C -2.0266,E1 24.8803,E2 311.8098} C_DIS
LIN {X -72.3616,Y 68.0556,Z 103,A 131.4769,B 24.9226,C -2.0315,E1 24.8843,E2 313.93} C_DIS
LIN {X -69.8005,Y 70.68,Z 103,A 129.35,B 24.9222,C -2.0363,E1 24.8885,E2 316.0548} C_DIS
LIN {X -67.1611,Y 73.1926,Z 103,A 127.2379,B 24.9219,C -2.0408,E1 24.8928,E2 318.1646} C_DIS
LIN {X -64.4315,Y 75.6066,Z 103,A 125.1816,B 24.9214,C -2.0471,E1 24.8971,E2 320.2139} C_DIS
LIN {X -62.0626,Y 77.5653,Z 103,A 123.2016,B 24.9217,C -2.044,E1 24.9014,E2 322.2089} C_DIS
LIN {X -58.9933,Y 79.9232,Z 103,A 121.0152,B 24.9212,C -2.0502,E1 24.9063,E2 324.3883} C_DIS
LIN {X -56.4758,Y 81.7211,Z 103,A 119.4218,B 24.9204,C -2.0603,E1 24.9099,E2 325.9632} C_DIS
LIN {X -53.8189,Y 83.4945,Z 103,A 117.4586,B 24.9204,C -2.0598,E1 24.9145,E2 327.9341} C_DIS
LIN {X -51.049,Y 85.218,Z 103,A 115.6793,B 24.9199,C -2.0667,E1 24.9187,E2 329.7023} C_DIS
LIN {X -48.9499,Y 86.4409,Z 103,A 114.2722,B 24.9197,C -2.069,E1 24.9221,E2 331.1082} C_DIS
LIN {X -46.4515,Y 87.807,Z 103,A 112.5216,B 24.9197,C -2.0681,E1 24.9264,E2 332.8659} C_DIS
LIN {X -43.5745,Y 89.2715,Z 103,A 110.5891,B 24.9197,C -2.0686,E1 24.9313,E2 334.8022} C_DIS
LIN {X -40.6503,Y 90.6386,Z 103,A 108.9118,B 24.919,C -2.0779,E1 24.9355,E2 336.4617} C_DIS
LIN {X -38.0123,Y 91.778,Z 103,A 107.2232,B 24.919,C -2.0791,E1 24.9398,E2 338.1512} C_DIS
LIN {X -35.9915,Y 92.5879,Z 103,A 105.7613,B 24.9194,C -2.0737,E1 24.9437,E2 339.6291} C_DIS
LIN {X -32.6904,Y 93.8038,Z 103,A 103.8682,B 24.9188,C -2.081,E1 24.9486,E2 341.5087} C_DIS
LIN {X -29.5915,Y 94.8269,Z 103,A 101.9413,B 24.9188,C -2.0817,E1 24.9537,E2 343.4374} C_DIS
LIN {X -26.8973,Y 95.6261,Z 103,A 100.3592,B 24.9185,C -2.0848,E1 24.958,E2 345.0147} C_DIS
LIN {X -24.1459,Y 96.3593,Z 103,A 98.608,B 24.9187,C -2.0826,E1 24.9627,E2 346.7738} C_DIS
LIN {X -21.0033,Y 97.091,Z 103,A 96.846,B 24.9183,C -2.0877,E1 24.9675,E2 348.5257} C_DIS
LIN {X -18.2145,Y 97.6542,Z 103,A 95.2643,B 24.918,C -2.0911,E1 24.9718,E2 350.1011} C_DIS
LIN {X -15.3556,Y 98.1428,Z 103,A 93.4859,B 24.9182,C -2.0886,E1 24.9767,E2 351.8871} C_DIS
LIN {X -12.154,Y 98.5922,Z 103,A 91.719,B 24.9178,C -2.0932,E1 24.9816,E2 353.6444} C_DIS
LIN {X -9.7359,Y 98.8603,Z 103,A 90.1481,B 24.9182,C -2.088,E1 24.986,E2 355.2287} C_DIS
LIN {X -6.514,Y 99.123,Z 103,A 88.3897,B 24.9179,C -2.0926,E1 24.9909,E2 356.9768} C_DIS
LIN {X -3.2256,Y 99.2845,Z 103,A 86.4472,B 24.9179,C -2.0917,E1 24.9963,E2 358.922} C_DIS
LIN {X 0.0054,Y 99.3385,Z 103,A 84.5174,B 24.9181,C -2.0897,E1 25.0017,E2 360.8565} C_DIS
LIN {X 3.2374,Y 99.2841,Z 103,A 82.817,B 24.9176,C -2.0958,E1 25.0064,E2 362.542} C_DIS
LIN {X 5.9921,Y 99.1571,Z 103,A 81.1179,B 24.9179,C -2.0919,E1 25.0112,E2 364.2497} C_DIS
LIN {X 9.4359,Y 98.888,Z 103,A 79.2409,B 24.9176,C -2.096,E1 25.0164,E2 366.1161} C_DIS
LIN {X 11.7672,Y 98.6375,Z 103,A 77.8884,B 24.9176,C -2.0958,E1 25.0201,E2 367.4682} C_DIS
LIN {X 14.598,Y 98.2599,Z 103,A 76.0758,B 24.9181,C -2.0893,E1 25.0252,E2 369.2946} C_DIS
LIN {X 17.7746,Y 97.7337,Z 103,A 74.381,B 24.9177,C -2.0946,E1 25.0298,E2 370.975} C_DIS
LIN {X 20.1546,Y 97.2708,Z 103,A 72.9134,B 24.918,C -2.0914,E1 25.0338,E2 372.4483} C_DIS
LIN {X 23.3747,Y 96.5475,Z 103,A 70.9827,B 24.9181,C -2.0894,E1 25.0391,E2 374.381} C_DIS
LIN {X 26.5003,Y 95.7386,Z 103,A 69.0582,B 24.9184,C -2.0859,E1 25.0443,E2 376.3109} C_DIS
LIN {X 29.5976,Y 94.8251,Z 103,A 67.3051,B 24.9182,C -2.0886,E1 25.0489,E2 378.0545} C_DIS
LIN {X 32.7179,Y 93.7942,Z 103,A 65.3704,B 24.9184,C -2.0855,E1 25.0541,E2 379.9927} C_DIS
LIN {X 35.7546,Y 92.6809,Z 103,A 63.6084,B 24.9183,C -2.0876,E1 25.0586,E2 381.7461} C_DIS
LIN {X 38.5761,Y 91.5405,Z 103,A 61.7397,B 24.9187,C -2.0815,E1 25.0635,E2 383.6248} C_DIS
LIN {X 41.3794,Y 90.3099,Z 103,A 59.9345,B 24.919,C -2.078,E1 25.0681,E2 385.4338} C_DIS
LIN {X 44.2854,Y 88.9191,Z 103,A 58.1855,B 24.9189,C -2.0798,E1 25.0725,E2 387.1738} C_DIS
LIN {X 47.2024,Y 87.4056,Z 103,A 56.2524,B 24.9192,C -2.0759,E1 25.0773,E2 389.1108} C_DIS
LIN {X 49.659,Y 86.0337,Z 103,A 54.7412,B 24.919,C -2.0778,E1 25.0809,E2 390.613} C_DIS
LIN {X 52.2902,Y 84.4611,Z 103,A 52.7752,B 24.9198,C -2.0677,E1 25.0856,E2 392.5968} C_DIS
LIN {X 55.5787,Y 82.3335,Z 103,A 50.651,B 24.9198,C -2.0692,E1 25.0906,E2 394.7105} C_DIS
LIN {X 58.176,Y 80.5213,Z 103,A 48.8973,B 24.9198,C -2.0688,E1 25.0946,E2 396.4589} C_DIS
LIN {X 60.6343,Y 78.6846,Z 103,A 47.0904,B 24.9201,C -2.0643,E1 25.0986,E2 398.27} C_DIS
LIN {X 63.328,Y 76.5335,Z 103,A 45.0595,B 24.9205,C -2.0589,E1 25.103,E2 400.3059} C_DIS
LIN {X 65.8136,Y 74.409,Z 103,A 43.0678,B 24.9211,C -2.0511,E1 25.1072,E2 402.3081} C_DIS
LIN {X 68.5011,Y 71.9427,Z 103,A 40.9712,B 24.9214,C -2.0471,E1 25.1115,E2 404.4057} C_DIS
LIN {X 70.9498,Y 69.5274,Z 103,A 39.0334,B 24.9216,C -2.0446,E1 25.1153,E2 406.3411} C_DIS
LIN {X 73.2704,Y 67.0764,Z 103,A 37.1966,B 24.9216,C -2.0446,E1 25.1188,E2 408.1701} C_DIS
LIN {X 75.6159,Y 64.4206,Z 103,A 35.157,B 24.922,C -2.04,E1 25.1225,E2 410.2111} C_DIS
LIN {X 77.8622,Y 61.6868,Z 103,A 33.0904,B 24.9224,C -2.0342,E1 25.1262,E2 412.282} C_DIS
LIN {X 80.0789,Y 58.7807,Z 103,A 31.039,B 24.9226,C -2.0312,E1 25.1296,E2 414.3306} C_DIS
LIN {X 81.6779,Y 56.5379,Z 103,A 29.474,B 24.9229,C -2.0281,E1 25.1321,E2 415.8952} C_DIS
LIN {X 83.4946,Y 53.8188,Z 103,A 27.5553,B 24.9233,C -2.022,E1 25.1351,E2 417.8189} C_DIS
LIN {X 84.9689,Y 51.4596,Z 103,A 25.9792,B 24.9236,C -2.0188,E1 25.1374,E2 419.3943} C_DIS
LIN {X 86.4449,Y 48.9427,Z 103,A 24.3905,B 24.9236,C -2.018,E1 25.1396,E2 420.9769} C_DIS
LIN {X 87.8078,Y 46.45,Z 103,A 22.6597,B 24.9243,C -2.0099,E1 25.1419,E2 422.7176} C_DIS
LIN {X 89.2691,Y 43.5793,Z 103,A 20.7516,B 24.9248,C -2.0027,E1 25.1443,E2 424.6325} C_DIS
LIN {X 90.6448,Y 40.6366,Z 103,A 19.0491,B 24.9247,C -2.0041,E1 25.1462,E2 426.3224} C_DIS
LIN {X 91.7756,Y 38.0182,Z 103,A 17.4141,B 24.925,C -1.9998,E1 25.148,E2 427.9588} C_DIS
LIN {X 92.6887,Y 35.734,Z 103,A 15.8438,B 24.9258,C -1.9896,E1 25.1496,E2 429.5442} C_DIS
LIN {X 93.7994,Y 32.7031,Z 103,A 14.098,B 24.9258,C -1.9887,E1 25.1513,E2 431.2825} C_DIS
LIN {X 94.7,Y 30.0009,Z 103,A 12.3204,B 24.9266,C -1.9784,E1 25.1528,E2 433.0743} C_DIS
LIN {X 95.6406,Y 26.8461,Z 103,A 10.5733,B 24.9266,C -1.9787,E1 25.1542,E2 434.8108} C_DIS
LIN {X 96.368,Y 24.1108,Z 103,A 8.8565,B 24.9272,C -1.9703,E1 25.1554,E2 436.5374} C_DIS
LIN {X 97.0901,Y 21.0075,Z 103,A 7.1269,B 24.9273,C -1.9689,E1 25.1564,E2 438.2603} C_DIS
LIN {X 97.6577,Y 18.1963,Z 103,A 5.5456,B 24.9275,C -1.9666,E1 25.1573,E2 439.8377} C_DIS
LIN {X 98.1357,Y 15.4017,Z 103,A 3.8097,B 24.9282,C -1.9575,E1 25.1581,E2 441.585} C_DIS
LIN {X 98.5907,Y 12.1657,Z 103,A 2.0493,B 24.9282,C -1.9564,E1 25.1587,E2 443.3375} C_DIS
LIN {X 98.8591,Y 9.7469,Z 103,A 0.4911,B 24.929,C -1.9458,E1 25.1591,E2 444.9115} C_DIS
LIN {X 99.1235,Y 6.5078,Z 103,A -1.2621,B 24.929,C -1.9447,E1 25.1595,E2 446.657} C_DIS
LIN {X 99.284,Y 3.2414,Z 103,A -3.1797,B 24.9296,C -1.9373,E1 25.1597,E2 448.5805} C_DIS
LIN {X 99.3379,Y 0.1213,Z 103,A -5.0402,B 24.9302,C -1.9291,E1 25.1597,E2 450.4494} C_DIS
LIN {X 99.2839,Y -3.2424,Z 103,A -6.8497,B 24.9303,C -1.9281,E1 25.1597,E2 452.2506} C_DIS
LIN {X 99.1234,Y -6.5081,Z 103,A -8.7661,B 24.9308,C -1.9208,E1 25.1594,E2 454.1728} C_DIS
LIN {X 98.8992,Y -9.3147,Z 103,A -10.2786,B 24.9308,C -1.92,E1 25.159,E2 455.6782} C_DIS
LIN {X 98.6413,Y -11.7348,Z 103,A -11.6725,B 24.9312,C -1.9158,E1 25.1586,E2 457.0737} C_DIS
LIN {X 98.292,Y -14.3745,Z 103,A -13.3969,B 24.9321,C -1.9033,E1 25.1579,E2 458.8173} C_DIS
LIN {X 97.7265,Y -17.8146,Z 103,A -15.1897,B 24.9319,C -1.9056,E1 25.157,E2 460.5943} C_DIS
LIN {X 97.2634,Y -20.1903,Z 103,A -16.6398,B 24.9324,C -1.8989,E1 25.1562,E2 462.0516} C_DIS
LIN {X 96.5493,Y -23.3674,Z 103,A -18.5231,B 24.9328,C -1.8927,E1 25.155,E2 463.9386} C_DIS
LIN {X 95.8512,Y -26.0836,Z 103,A -20.1094,B 24.9331,C -1.8888,E1 25.1539,E2 465.525} C_DIS
LIN {X 95.0584,Y -28.8452,Z 103,A -21.8609,B 24.9338,C -1.8798,E1 25.1525,E2 467.2878} C_DIS
LIN {X 94.068,Y -31.922,Z 103,A -23.6063,B 24.9338,C -1.8787,E1 25.151,E2 469.0259} C_DIS
LIN {X 93.2274,Y -34.3002,Z 103,A -25.2162,B 24.9346,C -1.868,E1 25.1494,E2 470.6519} C_DIS
LIN {X 91.9189,Y -37.6662,Z 103,A -27.0631,B 24.9344,C -1.871,E1 25.1476,E2 472.4816} C_DIS
LIN {X 90.8086,Y -40.2731,Z 103,A -28.6842,B 24.9347,C -1.8665,E1 25.1458,E2 474.1044} C_DIS
LIN {X 89.6198,Y -42.8498,Z 103,A -30.413,B 24.9353,C -1.858,E1 25.1437,E2 475.8441} C_DIS
LIN {X 88.187,Y -45.7294,Z 103,A -32.3238,B 24.9358,C -1.8502,E1 25.1413,E2 477.7631} C_DIS
LIN {X 86.638,Y -48.5969,Z 103,A -34.0249,B 24.9358,C -1.8518,E1 25.139,E2 479.4516} C_DIS
LIN {X 85.3078,Y -50.8972,Z 103,A -35.718,B 24.9365,C -1.841,E1 25.1366,E2 481.1614} C_DIS
LIN {X 83.4713,Y -53.8551,Z 103,A -37.6031,B 24.9365,C -1.8401,E1 25.1338,E2 483.039} C_DIS
LIN {X 81.9063,Y -56.2094,Z 103,A -39.1593,B 24.9366,C -1.8385,E1 25.1313,E2 484.5914} C_DIS
LIN {X 80.5152,Y -58.1845,Z 103,A -40.5546,B 24.9369,C -1.8346,E1 25.1291,E2 485.9891} C_DIS
LIN {X 79.0539,Y -60.155,Z 103,A -42.1691,B 24.9377,C -1.8229,E1 25.1263,E2 487.6236} C_DIS
LIN {X 76.7919,Y -63.0171,Z 103,A -44.262,B 24.9381,C -1.8177,E1 25.1227,E2 489.7189} C_DIS
LIN {X 74.5633,Y -65.6372,Z 103,A -46.0471,B 24.9379,C -1.8204,E1 25.1194,E2 491.4895} C_DIS
LIN {X 72.3582,Y -68.0593,Z 103,A -48.0075,B 24.9384,C -1.8129,E1 25.1157,E2 493.4592} C_DIS
LIN {X 69.8103,Y -70.6703,Z 103,A -50.0404,B 24.9386,C -1.8105,E1 25.1117,E2 495.489} C_DIS
Enddeposition()
END
